C09123=1121.889,263.715,-72.224,-178.349,10.071,149.559
C09124=1121.884,263.963,-72.253,-178.345,10.075,149.559
C09125=1121.880,264.212,-72.283,-178.342,10.077,149.559
C09126=1121.876,264.460,-72.312,-178.338,10.080,149.558
C09127=1121.872,264.708,-72.342,-178.335,10.083,149.558
C09128=1121.868,264.956,-72.371,-178.333,10.085,149.558
C09129=1121.863,265.205,-72.400,-178.330,10.088,149.558
C09130=1121.858,265.453,-72.429,-178.327,10.090,149.558
C09131=1121.854,265.701,-72.458,-178.325,10.093,149.558
C09132=1121.850,265.949,-72.488,-178.323,10.095,149.558
C09133=1121.846,266.198,-72.517,-178.320,10.098,149.558
C09134=1121.842,266.411,-72.542,-178.317,10.100,149.558
C09135=1121.839,266.625,-72.568,-178.315,10.102,149.558
C09136=1121.835,266.838,-72.593,-178.313,10.104,149.557
C09137=1121.832,267.051,-72.619,-178.310,10.106,149.557
C09138=1121.828,267.263,-72.643,-178.308,10.108,149.557
C09139=1121.824,267.477,-72.669,-178.306,10.110,149.557
C09140=1121.821,267.690,-72.694,-178.304,10.112,149.557
C09141=1121.817,267.904,-72.719,-178.302,10.114,149.557
C09142=1121.813,268.152,-72.748,-178.299,10.117,149.557
C09143=1121.809,268.400,-72.778,-178.296,10.119,149.557
C09144=1121.804,268.649,-72.808,-178.293,10.121,149.557
C09145=1121.800,268.897,-72.837,-178.290,10.124,149.557
C09146=1121.795,269.145,-72.867,-178.287,10.127,149.556
C09147=1121.791,269.393,-72.897,-178.285,10.130,149.556
C09148=1121.787,269.641,-72.926,-178.282,10.132,149.556
C09149=1121.783,269.890,-72.956,-178.279,10.134,149.556
C09150=1121.779,270.138,-72.985,-178.276,10.137,149.556
C09151=1121.775,270.386,-73.015,-178.273,10.140,149.556
C09152=1121.771,270.634,-73.044,-178.271,10.142,149.556
C09153=1121.766,270.883,-73.074,-178.268,10.145,149.556
C09154=1121.762,271.131,-73.105,-178.265,10.147,149.556
C09155=1121.758,271.379,-73.134,-178.262,10.150,149.555
C09156=1121.753,271.627,-73.163,-178.259,10.153,149.555
C09157=1121.749,271.875,-73.193,-178.257,10.155,149.555
C09158=1121.745,272.124,-73.222,-178.254,10.158,149.555
C09159=1121.741,272.371,-73.252,-178.251,10.160,149.555
C09160=1121.737,272.620,-73.282,-178.248,10.163,149.555
C09161=1121.732,272.868,-73.312,-178.245,10.166,149.555
C09162=1121.728,273.116,-73.342,-178.242,10.169,149.555
C09163=1121.724,273.364,-73.372,-178.239,10.171,149.555
C09164=1121.720,273.612,-73.401,-178.236,10.174,149.554
C09165=1121.715,273.860,-73.432,-178.233,10.177,149.554
C09166=1121.711,274.109,-73.461,-178.230,10.179,149.554
C09167=1121.707,274.357,-73.491,-178.227,10.182,149.554
C09168=1121.703,274.604,-73.521,-178.224,10.185,149.554
C09169=1121.699,274.853,-73.551,-178.221,10.188,149.554
C09170=1121.694,275.102,-73.581,-178.218,10.190,149.554
C09171=1121.691,275.350,-73.611,-178.215,10.193,149.553
C09172=1121.686,275.598,-73.640,-178.212,10.196,149.553
C09173=1121.682,275.846,-73.671,-178.209,10.198,149.553
C09174=1121.678,276.094,-73.701,-178.206,10.201,149.553
C09175=1121.674,276.342,-73.731,-178.203,10.204,149.553
C09176=1121.669,276.590,-73.761,-178.200,10.206,149.553
C09177=1121.665,276.838,-73.791,-178.197,10.209,149.553
C09178=1121.661,277.087,-73.821,-178.194,10.211,149.552
C09179=1121.657,277.335,-73.852,-178.191,10.214,149.552
C09180=1121.653,277.583,-73.881,-178.188,10.217,149.552
C09181=1121.649,277.831,-73.911,-178.184,10.219,149.552
C09182=1121.644,278.079,-73.941,-178.182,10.222,149.552
C09183=1121.640,278.327,-73.971,-178.178,10.225,149.552
C09184=1121.637,278.575,-74.002,-178.175,10.228,149.551
C09185=1121.632,278.824,-74.032,-178.171,10.231,149.551
C09186=1121.628,279.072,-74.062,-178.168,10.233,149.551
C09187=1121.623,279.320,-74.093,-178.165,10.236,149.551
C09188=1121.619,279.568,-74.122,-178.162,10.238,149.551
C09189=1121.615,279.817,-74.154,-178.158,10.242,149.551
C09190=1121.612,280.029,-74.179,-178.156,10.244,149.550
C09191=1121.608,280.243,-74.205,-178.153,10.246,149.550
C09192=1121.604,280.456,-74.231,-178.151,10.248,149.550
C09193=1121.601,280.669,-74.257,-178.147,10.251,149.550
C09194=1121.597,280.882,-74.283,-178.144,10.254,149.550
C09195=1121.594,281.095,-74.309,-178.142,10.255,149.549
C09196=1121.590,281.308,-74.336,-178.139,10.258,149.549
C09197=1121.583,281.692,-74.383,-178.134,10.262,149.549
C09198=1121.579,281.940,-74.413,-178.131,10.264,149.549
C09199=1121.575,282.189,-74.444,-178.128,10.267,149.549
C09200=1121.571,282.437,-74.475,-178.124,10.270,149.548
C09201=1121.567,282.685,-74.504,-178.121,10.272,149.548
C09202=1121.562,282.933,-74.535,-178.119,10.275,149.548
C09203=1121.559,283.181,-74.565,-178.115,10.277,149.548
C09204=1121.554,283.429,-74.596,-178.113,10.279,149.548
C09205=1121.550,283.677,-74.626,-178.110,10.282,149.548
C09206=1121.546,283.925,-74.657,-178.107,10.285,149.547
C09207=1121.542,284.173,-74.688,-178.103,10.287,149.547
C09208=1121.538,284.421,-74.718,-178.100,10.290,149.547
C09209=1121.533,284.669,-74.749,-178.097,10.293,149.547
C09210=1121.529,284.918,-74.780,-178.094,10.295,149.547
C09211=1121.525,285.165,-74.810,-178.091,10.298,149.547
C09212=1121.521,285.413,-74.841,-178.088,10.300,149.546
C09213=1121.517,285.662,-74.872,-178.085,10.303,149.546
C09214=1121.513,285.910,-74.902,-178.082,10.305,149.546
C09215=1121.508,286.158,-74.933,-178.079,10.307,149.546
C09216=1121.504,286.406,-74.964,-178.076,10.310,149.546
C09217=1121.500,286.654,-74.995,-178.073,10.313,149.546
C09218=1121.496,286.902,-75.025,-178.070,10.315,149.545
C09219=1121.492,287.150,-75.056,-178.067,10.318,149.545
C09220=1121.488,287.398,-75.087,-178.064,10.320,149.545
C09221=1121.483,287.646,-75.117,-178.060,10.323,149.545
C09222=1121.479,287.894,-75.149,-178.057,10.326,149.545
C09223=1121.475,288.142,-75.180,-178.055,10.327,149.544
C09224=1121.471,288.390,-75.210,-178.052,10.330,149.544
C09225=1121.467,288.638,-75.241,-178.049,10.333,149.544
C09226=1121.462,288.886,-75.272,-178.045,10.335,149.544
C09227=1121.458,289.135,-75.303,-178.043,10.338,149.544
C09228=1121.455,289.382,-75.334,-178.039,10.340,149.544
C09229=1121.451,289.631,-75.365,-178.036,10.343,149.543
C09230=1121.446,289.879,-75.396,-178.033,10.346,149.543
C09231=1121.441,290.127,-75.427,-178.030,10.348,149.543
C09232=1121.438,290.375,-75.459,-178.027,10.351,149.543
C09233=1121.433,290.623,-75.489,-178.024,10.353,149.543
C09234=1121.430,290.871,-75.520,-178.021,10.356,149.543
C09235=1121.426,291.118,-75.551,-178.018,10.358,149.542
C09236=1121.422,291.367,-75.582,-178.015,10.361,149.542
C09237=1121.417,291.615,-75.613,-178.012,10.363,149.542
C09238=1121.413,291.863,-75.645,-178.009,10.366,149.542
C09239=1121.409,292.111,-75.676,-178.006,10.368,149.542
C09240=1121.405,292.360,-75.707,-178.003,10.371,149.542
C09241=1121.401,292.607,-75.738,-177.999,10.374,149.541
C09242=1121.397,292.855,-75.769,-177.996,10.376,149.541
C09243=1121.393,293.103,-75.800,-177.994,10.378,149.541
C09244=1121.389,293.351,-75.832,-177.991,10.381,149.541
C09245=1121.384,293.599,-75.863,-177.987,10.383,149.541
C09246=1121.378,293.982,-75.912,-177.983,10.387,149.540
C09247=1121.371,294.365,-75.959,-177.978,10.391,149.540
C09248=1121.365,294.749,-76.008,-177.974,10.395,149.540
C09249=1121.359,295.132,-76.056,-177.969,10.399,149.539
C09250=1121.354,295.379,-76.088,-177.966,10.401,149.539
C09251=1121.351,295.627,-76.119,-177.962,10.404,149.539
C09252=1121.346,295.875,-76.150,-177.959,10.407,149.539
C09253=1121.342,296.123,-76.182,-177.956,10.409,149.539
C09254=1121.338,296.372,-76.213,-177.953,10.412,149.539
C09255=1121.334,296.619,-76.245,-177.950,10.414,149.538
C09256=1121.330,296.868,-76.277,-177.947,10.417,149.538
C09257=1121.326,297.115,-76.307,-177.943,10.419,149.538
C09258=1121.322,297.364,-76.339,-177.941,10.422,149.538
C09259=1121.318,297.611,-76.371,-177.938,10.424,149.538
C09260=1121.313,297.860,-76.402,-177.935,10.427,149.538
C09261=1121.309,298.108,-76.434,-177.932,10.429,149.537
C09262=1121.305,298.355,-76.466,-177.929,10.432,149.537
C09263=1121.301,298.604,-76.497,-177.925,10.434,149.537
C09264=1121.297,298.851,-76.528,-177.922,10.437,149.537
C09265=1121.293,299.099,-76.560,-177.919,10.439,149.537
C09266=1121.289,299.347,-76.592,-177.916,10.442,149.537
C09267=1121.285,299.595,-76.623,-177.913,10.445,149.536
C09268=1121.280,299.844,-76.655,-177.910,10.447,149.536
C09269=1121.277,300.092,-76.687,-177.906,10.450,149.536
C09270=1121.272,300.339,-76.719,-177.904,10.452,149.536
C09271=1121.269,300.587,-76.750,-177.901,10.454,149.536
C09272=1121.265,300.835,-76.782,-177.898,10.457,149.535
C09273=1121.260,301.083,-76.814,-177.895,10.459,149.535
C09274=1121.256,301.331,-76.846,-177.892,10.462,149.535
C09275=1121.252,301.579,-76.877,-177.888,10.465,149.535
C09276=1121.248,301.827,-76.909,-177.885,10.467,149.535
C09277=1121.243,302.075,-76.941,-177.882,10.470,149.534
C09278=1121.240,302.323,-76.973,-177.879,10.473,149.534
C09279=1121.235,302.570,-77.004,-177.876,10.475,149.534
C09280=1121.232,302.818,-77.036,-177.873,10.478,149.534
C09281=1121.227,303.067,-77.069,-177.870,10.480,149.534
C09282=1121.223,303.314,-77.100,-177.867,10.482,149.534
C09283=1121.219,303.562,-77.132,-177.864,10.485,149.533
C09284=1121.215,303.811,-77.165,-177.861,10.487,149.533
C09285=1121.210,304.058,-77.196,-177.858,10.490,149.533
C09286=1121.207,304.306,-77.228,-177.855,10.493,149.533
C09287=1121.202,304.554,-77.260,-177.851,10.495,149.533
C09288=1121.199,304.802,-77.293,-177.848,10.498,149.533
C09289=1121.195,305.049,-77.324,-177.845,10.500,149.532
C09290=1121.190,305.297,-77.357,-177.842,10.503,149.532
C09291=1121.186,305.545,-77.389,-177.839,10.506,149.532
C09292=1121.182,305.794,-77.421,-177.836,10.508,149.532
C09293=1121.178,306.041,-77.453,-177.833,10.510,149.532
C09294=1121.174,306.289,-77.484,-177.830,10.512,149.531
C09295=1121.170,306.537,-77.518,-177.827,10.515,149.531
C09296=1121.166,306.785,-77.549,-177.824,10.518,149.531
C09297=1121.162,307.033,-77.582,-177.821,10.520,149.531
C09298=1121.158,307.246,-77.609,-177.818,10.522,149.531
C09299=1121.155,307.459,-77.637,-177.815,10.525,149.531
C09300=1121.151,307.671,-77.664,-177.813,10.527,149.531
C09301=1121.148,307.884,-77.693,-177.809,10.529,149.530
C09302=1121.144,308.097,-77.720,-177.807,10.531,149.530
C09303=1121.141,308.310,-77.747,-177.805,10.533,149.530
C09304=1121.137,308.522,-77.775,-177.802,10.536,149.530
C09305=1121.133,308.736,-77.803,-177.799,10.538,149.530
C09306=1121.130,308.983,-77.835,-177.796,10.540,149.530
C09307=1121.125,309.232,-77.868,-177.793,10.543,149.529
C09308=1121.121,309.479,-77.899,-177.790,10.545,149.529
C09309=1121.117,309.727,-77.933,-177.787,10.548,149.529
C09310=1121.113,309.975,-77.964,-177.783,10.550,149.529
C09311=1121.109,310.223,-77.998,-177.780,10.553,149.529
C09312=1121.105,310.471,-78.029,-177.778,10.555,149.528
C09313=1121.101,310.719,-78.062,-177.775,10.558,149.528
C09314=1121.098,310.966,-78.094,-177.771,10.560,149.528
C09315=1121.093,311.214,-78.126,-177.768,10.563,149.528
C09316=1121.088,311.462,-78.160,-177.765,10.565,149.528
C09317=1121.085,311.710,-78.191,-177.762,10.568,149.528
C09318=1121.081,311.958,-78.225,-177.759,10.571,149.527
C09319=1121.077,312.206,-78.256,-177.756,10.573,149.527
C09320=1121.073,312.453,-78.290,-177.753,10.576,149.527
C09321=1121.068,312.702,-78.322,-177.749,10.578,149.527
C09322=1121.065,312.949,-78.355,-177.746,10.581,149.527
C09323=1121.061,313.197,-78.388,-177.743,10.583,149.527
C09324=1121.057,313.445,-78.420,-177.740,10.586,149.526
C09325=1121.053,313.693,-78.453,-177.738,10.588,149.526
C09326=1121.048,313.941,-78.485,-177.734,10.590,149.526
C09327=1121.044,314.188,-78.517,-177.731,10.593,149.526
C09328=1121.040,314.435,-78.551,-177.728,10.595,149.526
C09329=1121.036,314.684,-78.583,-177.725,10.598,149.525
C09330=1121.032,314.931,-78.616,-177.722,10.601,149.525
C09331=1121.028,315.179,-78.649,-177.718,10.603,149.525
C09332=1121.024,315.427,-78.681,-177.715,10.606,149.525
C09333=1121.020,315.675,-78.714,-177.712,10.608,149.525
C09334=1121.016,315.922,-78.747,-177.709,10.611,149.524
C09335=1121.012,316.171,-78.779,-177.706,10.614,149.524
C09336=1121.008,316.418,-78.812,-177.703,10.616,149.524
C09337=1121.004,316.666,-78.846,-177.700,10.618,149.524
C09338=1121.000,316.914,-78.878,-177.697,10.620,149.524
C09339=1120.996,317.161,-78.911,-177.694,10.623,149.524
C09340=1120.992,317.410,-78.944,-177.691,10.626,149.523
C09341=1120.988,317.657,-78.977,-177.687,10.628,149.523
C09342=1120.984,317.905,-79.009,-177.684,10.631,149.523
C09343=1120.980,318.153,-79.043,-177.681,10.633,149.523
C09344=1120.976,318.401,-79.076,-177.678,10.636,149.523
C09345=1120.972,318.649,-79.109,-177.674,10.638,149.522
C09346=1120.968,318.896,-79.142,-177.671,10.641,149.522
C09347=1120.964,319.144,-79.176,-177.668,10.643,149.522
C09348=1120.960,319.392,-79.207,-177.665,10.646,149.522
C09349=1120.956,319.640,-79.241,-177.662,10.649,149.522
C09350=1120.952,319.888,-79.274,-177.659,10.650,149.521
C09351=1120.948,320.135,-79.307,-177.656,10.653,149.521
C09352=1120.944,320.383,-79.340,-177.653,10.656,149.521
C09353=1120.940,320.631,-79.373,-177.650,10.658,149.521
C09354=1120.937,320.843,-79.402,-177.647,10.661,149.521
C09355=1120.933,321.056,-79.430,-177.644,10.663,149.521
C09356=1120.929,321.268,-79.459,-177.642,10.664,149.520
C09357=1120.926,321.481,-79.487,-177.639,10.667,149.520
C09358=1120.923,321.694,-79.516,-177.636,10.669,149.520
C09359=1120.920,321.907,-79.544,-177.634,10.671,149.520
C09360=1120.916,322.120,-79.573,-177.631,10.674,149.520
C09361=1120.912,322.332,-79.601,-177.628,10.675,149.520
C09362=1120.909,322.581,-79.635,-177.625,10.678,149.520
C09363=1120.905,322.828,-79.668,-177.622,10.680,149.519
C09364=1120.901,323.075,-79.702,-177.619,10.683,149.519
C09365=1120.897,323.323,-79.735,-177.616,10.686,149.519
C09366=1120.892,323.571,-79.768,-177.612,10.688,149.519
C09367=1120.888,323.819,-79.801,-177.609,10.691,149.519
C09368=1120.885,324.067,-79.835,-177.606,10.693,149.518
C09369=1120.881,324.314,-79.868,-177.603,10.696,149.518
C09370=1120.877,324.562,-79.902,-177.599,10.698,149.518
C09371=1120.873,324.810,-79.935,-177.597,10.701,149.518
C09372=1120.868,325.057,-79.968,-177.594,10.703,149.518
C09373=1120.865,325.304,-80.002,-177.591,10.705,149.517
C09374=1120.861,325.553,-80.035,-177.588,10.708,149.517
C09375=1120.857,325.801,-80.069,-177.584,10.710,149.517
C09376=1120.853,326.048,-80.102,-177.581,10.713,149.517
C09377=1120.849,326.295,-80.136,-177.578,10.716,149.517
C09378=1120.845,326.543,-80.169,-177.575,10.718,149.517
C09379=1120.841,326.792,-80.202,-177.571,10.721,149.516
C09380=1120.837,327.039,-80.237,-177.568,10.723,149.516
C09381=1120.833,327.287,-80.270,-177.565,10.726,149.516
C09382=1120.829,327.534,-80.304,-177.562,10.728,149.516
C09383=1120.825,327.782,-80.337,-177.559,10.731,149.515
C09384=1120.821,328.030,-80.370,-177.556,10.733,149.515
C09385=1120.817,328.277,-80.404,-177.553,10.735,149.515
C09386=1120.812,328.525,-80.438,-177.550,10.738,149.515
C09387=1120.809,328.773,-80.472,-177.547,10.740,149.515
C09388=1120.805,329.021,-80.505,-177.543,10.743,149.515
C09389=1120.801,329.268,-80.539,-177.540,10.745,149.514
C09390=1120.797,329.516,-80.572,-177.537,10.748,149.514
C09391=1120.793,329.764,-80.607,-177.534,10.750,149.514
C09392=1120.789,330.011,-80.640,-177.530,10.753,149.514
C09393=1120.785,330.259,-80.674,-177.527,10.755,149.514
C09394=1120.782,330.507,-80.708,-177.524,10.758,149.514
C09395=1120.777,330.754,-80.742,-177.521,10.761,149.513
C09396=1120.773,331.001,-80.776,-177.518,10.763,149.513
C09397=1120.770,331.250,-80.810,-177.515,10.766,149.513
C09398=1120.766,331.497,-80.844,-177.511,10.768,149.513
C09399=1120.761,331.745,-80.877,-177.508,10.771,149.512
C09400=1120.758,331.993,-80.912,-177.505,10.772,149.512
C09401=1120.754,332.240,-80.945,-177.502,10.775,149.512
C09402=1120.749,332.488,-80.979,-177.499,10.778,149.512
C09403=1120.746,332.736,-81.013,-177.496,10.780,149.512
C09404=1120.742,332.983,-81.047,-177.493,10.783,149.512
C09405=1120.737,333.230,-81.082,-177.490,10.785,149.511
C09406=1120.734,333.479,-81.115,-177.486,10.788,149.511
C09407=1120.730,333.726,-81.149,-177.483,10.790,149.511
C09408=1120.725,333.973,-81.184,-177.480,10.793,149.511
C09409=1120.722,334.221,-81.218,-177.477,10.795,149.511
C09410=1120.719,334.434,-81.247,-177.474,10.797,149.510
C09411=1120.715,334.646,-81.276,-177.471,10.800,149.510
C09412=1120.712,334.859,-81.305,-177.468,10.802,149.510
C09413=1120.709,335.071,-81.335,-177.466,10.804,149.510
C09414=1120.705,335.284,-81.364,-177.463,10.806,149.510
C09415=1120.702,335.497,-81.393,-177.460,10.808,149.510
C09416=1120.698,335.709,-81.422,-177.458,10.810,149.509
C09417=1120.695,335.922,-81.452,-177.455,10.812,149.509
C09418=1120.691,336.169,-81.486,-177.452,10.815,149.509
C09419=1120.687,336.417,-81.520,-177.448,10.817,149.509
C09420=1120.683,336.664,-81.555,-177.445,10.820,149.509
C09421=1120.679,336.911,-81.589,-177.442,10.823,149.509
C09422=1120.675,337.160,-81.624,-177.439,10.824,149.508
C09423=1120.671,337.407,-81.658,-177.436,10.827,149.508
C09424=1120.667,337.655,-81.692,-177.433,10.830,149.508
C09425=1120.663,337.902,-81.726,-177.430,10.832,149.508
C09426=1120.660,338.150,-81.761,-177.426,10.834,149.507
C09427=1120.656,338.397,-81.795,-177.423,10.837,149.507
C09428=1120.652,338.645,-81.830,-177.420,10.839,149.507
C09429=1120.647,338.893,-81.864,-177.417,10.842,149.507
C09430=1120.644,339.140,-81.898,-177.414,10.845,149.507
C09431=1120.639,339.388,-81.933,-177.410,10.847,149.506
C09432=1120.636,339.636,-81.967,-177.407,10.849,149.506
C09433=1120.632,339.883,-82.002,-177.404,10.852,149.506
C09434=1120.628,340.131,-82.036,-177.401,10.855,149.506
C09435=1120.624,340.378,-82.070,-177.397,10.857,149.506
C09436=1120.620,340.626,-82.105,-177.394,10.860,149.506
C09437=1120.616,340.873,-82.140,-177.391,10.861,149.505
C09438=1120.612,341.121,-82.175,-177.388,10.864,149.505
C09439=1120.608,341.368,-82.209,-177.385,10.867,149.505
C09440=1120.604,341.616,-82.243,-177.382,10.869,149.505
C09441=1120.600,341.864,-82.278,-177.378,10.871,149.504
C09442=1120.596,342.111,-82.313,-177.375,10.874,149.504
C09443=1120.592,342.358,-82.347,-177.372,10.877,149.504
C09444=1120.588,342.606,-82.382,-177.369,10.879,149.504
C09445=1120.584,342.854,-82.416,-177.366,10.882,149.504
C09446=1120.580,343.101,-82.452,-177.362,10.884,149.504
C09447=1120.577,343.349,-82.486,-177.359,10.887,149.503
C09448=1120.572,343.597,-82.521,-177.356,10.889,149.503
C09449=1120.569,343.844,-82.556,-177.353,10.892,149.503
C09450=1120.564,344.092,-82.591,-177.349,10.894,149.503
C09451=1120.561,344.339,-82.625,-177.346,10.897,149.503
C09452=1120.557,344.587,-82.661,-177.343,10.898,149.502
C09453=1120.553,344.834,-82.695,-177.340,10.901,149.502
C09454=1120.549,345.082,-82.730,-177.337,10.904,149.502
C09455=1120.545,345.329,-82.764,-177.334,10.906,149.502
C09456=1120.541,345.577,-82.799,-177.331,10.909,149.502
C09457=1120.538,345.824,-82.835,-177.327,10.911,149.501
C09458=1120.533,346.072,-82.869,-177.324,10.913,149.501
C09459=1120.529,346.319,-82.905,-177.321,10.916,149.501
C09460=1120.526,346.567,-82.939,-177.318,10.919,149.501
C09461=1120.522,346.814,-82.974,-177.314,10.921,149.501
C09462=1120.518,347.062,-83.009,-177.311,10.924,149.500
C09463=1120.514,347.309,-83.044,-177.308,10.926,149.500
C09464=1120.510,347.557,-83.079,-177.305,10.929,149.500
C09465=1120.506,347.805,-83.115,-177.301,10.931,149.500
C09466=1120.503,348.017,-83.144,-177.299,10.933,149.500
C09467=1120.499,348.229,-83.174,-177.296,10.935,149.499
C09468=1120.496,348.441,-83.205,-177.293,10.937,149.499
C09469=1120.493,348.654,-83.235,-177.291,10.939,149.499
C09470=1120.489,348.867,-83.265,-177.288,10.941,149.499
C09471=1120.486,349.079,-83.294,-177.285,10.944,149.499
C09472=1120.482,349.291,-83.325,-177.282,10.945,149.498
C09473=1120.480,349.504,-83.355,-177.279,10.948,149.498
C09474=1120.476,349.750,-83.391,-177.276,10.950,149.498
C09475=1120.472,349.999,-83.425,-177.272,10.953,149.498
C09476=1120.468,350.246,-83.461,-177.269,10.955,149.498
C09477=1120.464,350.494,-83.496,-177.266,10.958,149.497
C09478=1120.460,350.741,-83.531,-177.262,10.961,149.497
C09479=1120.456,350.989,-83.566,-177.259,10.963,149.497
C09480=1120.452,351.236,-83.602,-177.255,10.966,149.497
C09481=1120.449,351.484,-83.638,-177.252,10.968,149.496
C09482=1120.445,351.730,-83.673,-177.248,10.970,149.496
C09483=1120.441,351.978,-83.708,-177.244,10.974,149.496
C09484=1120.437,352.226,-83.743,-177.241,10.976,149.496
C09485=1120.433,352.473,-83.779,-177.238,10.979,149.495
C09486=1120.429,352.720,-83.814,-177.234,10.981,149.495
C09487=1120.425,352.968,-83.849,-177.231,10.983,149.495
C09488=1120.422,353.215,-83.885,-177.228,10.986,149.495
C09489=1120.418,353.463,-83.921,-177.223,10.989,149.494
C09490=1120.414,353.711,-83.957,-177.220,10.991,149.494
C09491=1120.409,353.957,-83.992,-177.217,10.994,149.494
C09492=1120.406,354.205,-84.027,-177.213,10.996,149.494
C09493=1120.402,354.453,-84.062,-177.210,10.999,149.493
C09494=1120.398,354.700,-84.098,-177.206,11.001,149.493
C09495=1120.394,354.948,-84.133,-177.203,11.003,149.493
C09496=1120.391,355.195,-84.169,-177.200,11.006,149.493
C09497=1120.387,355.442,-84.205,-177.197,11.008,149.492
C09498=1120.383,355.689,-84.240,-177.193,11.011,149.492
C09499=1120.379,355.937,-84.276,-177.189,11.014,149.492
C09500=1120.375,356.184,-84.312,-177.186,11.016,149.492
C09501=1120.371,356.432,-84.348,-177.182,11.019,149.491
C09502=1120.368,356.679,-84.383,-177.179,11.021,149.491
C09503=1120.364,356.927,-84.419,-177.176,11.023,149.491
C09504=1120.360,357.175,-84.455,-177.172,11.026,149.491
C09505=1120.356,357.422,-84.490,-177.169,11.028,149.490
C09506=1120.353,357.669,-84.527,-177.165,11.031,149.490
C09507=1120.348,357.916,-84.562,-177.162,11.033,149.490
C09508=1120.345,358.163,-84.597,-177.158,11.035,149.489
C09509=1120.340,358.411,-84.633,-177.155,11.038,149.489
C09510=1120.337,358.659,-84.669,-177.152,11.040,149.489
C09511=1120.333,358.906,-84.705,-177.148,11.043,149.489
C09512=1120.330,359.153,-84.741,-177.145,11.045,149.489
C09513=1120.325,359.401,-84.777,-177.141,11.047,149.488
C09514=1120.322,359.648,-84.813,-177.138,11.050,149.488
C09515=1120.318,359.895,-84.849,-177.135,11.052,149.488
C09516=1120.314,360.143,-84.885,-177.131,11.055,149.488
C09517=1120.310,360.391,-84.920,-177.128,11.057,149.487
C09518=1120.307,360.638,-84.957,-177.124,11.059,149.487
C09519=1120.302,360.885,-84.993,-177.121,11.062,149.487
C09520=1120.299,361.132,-85.029,-177.118,11.064,149.486
C09521=1120.295,361.380,-85.065,-177.115,11.067,149.486
C09522=1120.292,361.592,-85.096,-177.111,11.069,149.486
C09523=1120.289,361.804,-85.127,-177.109,11.071,149.486
C09524=1120.285,362.016,-85.158,-177.105,11.073,149.486
C09525=1120.282,362.229,-85.189,-177.103,11.075,149.485
C09526=1120.279,362.441,-85.219,-177.100,11.077,149.485
C09527=1120.276,362.653,-85.251,-177.097,11.079,149.485
C09528=1120.272,362.865,-85.282,-177.094,11.081,149.485
C09529=1120.269,363.078,-85.313,-177.091,11.083,149.484
C09530=1120.266,363.325,-85.348,-177.087,11.086,149.484
C09531=1120.262,363.572,-85.385,-177.084,11.088,149.484
C09532=1120.258,363.819,-85.421,-177.081,11.091,149.484
C09533=1120.254,364.067,-85.458,-177.077,11.093,149.484
C09534=1120.250,364.314,-85.494,-177.074,11.094,149.483
C09535=1120.246,364.562,-85.530,-177.071,11.097,149.483
C09536=1120.243,364.809,-85.566,-177.068,11.099,149.483
C09537=1120.239,365.056,-85.603,-177.064,11.102,149.482
C09538=1120.235,365.303,-85.639,-177.061,11.104,149.482
C09539=1120.231,365.551,-85.676,-177.057,11.106,149.482
C09540=1120.227,365.798,-85.711,-177.054,11.109,149.482
C09541=1120.224,366.046,-85.748,-177.051,11.111,149.481
C09542=1120.220,366.293,-85.785,-177.048,11.114,149.481
C09543=1120.216,366.540,-85.821,-177.044,11.116,149.481
C09544=1120.213,366.788,-85.857,-177.041,11.119,149.481
C09545=1120.208,367.035,-85.894,-177.038,11.121,149.481
C09546=1120.204,367.282,-85.931,-177.034,11.123,149.480
C09547=1120.201,367.529,-85.967,-177.031,11.126,149.480
C09548=1120.197,367.777,-86.003,-177.028,11.128,149.480
C09549=1120.193,368.024,-86.039,-177.025,11.130,149.480
C09550=1120.190,368.271,-86.077,-177.021,11.133,149.479
C09551=1120.186,368.519,-86.113,-177.018,11.135,149.479
C09552=1120.182,368.766,-86.150,-177.015,11.138,149.479
C09553=1120.178,369.013,-86.186,-177.011,11.140,149.479
C09554=1120.175,369.260,-86.222,-177.008,11.142,149.478
C09555=1120.170,369.507,-86.259,-177.005,11.145,149.478
C09556=1120.167,369.755,-86.296,-177.001,11.147,149.478
C09557=1120.164,370.002,-86.332,-176.998,11.149,149.478
C09558=1120.160,370.249,-86.369,-176.995,11.151,149.477
C09559=1120.155,370.497,-86.406,-176.992,11.154,149.477
C09560=1120.151,370.744,-86.443,-176.989,11.156,149.477
C09561=1120.149,370.991,-86.480,-176.985,11.159,149.477
C09562=1120.144,371.239,-86.517,-176.982,11.161,149.477
C09563=1120.140,371.486,-86.553,-176.979,11.164,149.476
C09564=1120.137,371.733,-86.590,-176.975,11.166,149.476
C09565=1120.133,371.980,-86.627,-176.972,11.169,149.476
C09566=1120.129,372.228,-86.664,-176.969,11.170,149.476
C09567=1120.125,372.475,-86.701,-176.966,11.173,149.476
C09568=1120.122,372.722,-86.737,-176.963,11.175,149.475
C09569=1120.118,372.969,-86.774,-176.960,11.178,149.475
C09570=1120.114,373.217,-86.811,-176.956,11.180,149.475
C09571=1120.110,373.464,-86.848,-176.953,11.183,149.475
C09572=1120.107,373.711,-86.884,-176.950,11.186,149.475
C09573=1120.103,373.957,-86.922,-176.947,11.187,149.474
C09574=1120.100,374.205,-86.959,-176.944,11.190,149.474
C09575=1120.096,374.453,-86.996,-176.941,11.192,149.474
C09576=1120.091,374.700,-87.033,-176.937,11.195,149.474
C09577=1120.087,374.947,-87.069,-176.934,11.197,149.474
C09578=1120.085,375.159,-87.101,-176.932,11.199,149.473
C09579=1120.082,375.371,-87.133,-176.929,11.202,149.473
C09580=1120.078,375.583,-87.164,-176.926,11.203,149.473
C09581=1120.075,375.795,-87.197,-176.924,11.205,149.473
C09582=1120.072,376.007,-87.229,-176.921,11.207,149.473
C09583=1120.069,376.220,-87.260,-176.918,11.210,149.473
C09584=1120.066,376.431,-87.292,-176.915,11.212,149.473
C09585=1120.062,376.644,-87.324,-176.913,11.214,149.473
C09586=1120.058,376.891,-87.361,-176.910,11.216,149.472
C09587=1120.055,377.139,-87.398,-176.907,11.219,149.472
C09588=1120.052,377.385,-87.435,-176.903,11.221,149.472
C09589=1120.047,377.632,-87.472,-176.900,11.224,149.472
C09590=1120.044,377.880,-87.510,-176.897,11.226,149.472
C09591=1120.040,378.127,-87.547,-176.894,11.229,149.471
C09592=1120.036,378.374,-87.584,-176.891,11.231,149.471
C09593=1120.033,378.621,-87.622,-176.888,11.233,149.471
C09594=1120.029,378.868,-87.659,-176.885,11.236,149.471
C09595=1120.025,379.115,-87.696,-176.882,11.239,149.471
C09596=1120.022,379.363,-87.734,-176.879,11.241,149.471
C09597=1120.017,379.610,-87.770,-176.875,11.244,149.471
C09598=1120.014,379.857,-87.808,-176.873,11.246,149.471
C09599=1120.010,380.104,-87.845,-176.870,11.248,149.470
C09600=1120.006,380.351,-87.883,-176.867,11.251,149.470
C09601=1120.003,380.599,-87.920,-176.864,11.253,149.470
C09602=1119.999,380.845,-87.958,-176.860,11.256,149.470
C09603=1119.996,381.093,-87.995,-176.857,11.259,149.470
C09604=1119.992,381.340,-88.032,-176.854,11.261,149.470
C09605=1119.987,381.587,-88.071,-176.852,11.263,149.470
C09606=1119.984,381.835,-88.108,-176.849,11.266,149.470
C09607=1119.980,382.081,-88.145,-176.846,11.269,149.469
C09608=1119.976,382.329,-88.183,-176.842,11.271,149.469
C09609=1119.973,382.576,-88.220,-176.840,11.274,149.469
C09610=1119.969,382.823,-88.258,-176.837,11.277,149.469
C09611=1119.965,383.070,-88.295,-176.833,11.279,149.469
C09612=1119.962,383.317,-88.333,-176.831,11.281,149.469
C09613=1119.958,383.564,-88.370,-176.828,11.284,149.469
C09614=1119.954,383.811,-88.407,-176.826,11.286,149.469
C09615=1119.950,384.059,-88.446,-176.824,11.288,149.469
C09616=1119.947,384.305,-88.483,-176.822,11.290,149.469
C09617=1119.943,384.553,-88.521,-176.820,11.293,149.469
C09618=1119.939,384.800,-88.558,-176.818,11.295,149.469
C09619=1119.936,385.047,-88.596,-176.816,11.297,149.469
C09620=1119.932,385.294,-88.634,-176.813,11.299,149.469
C09621=1119.928,385.541,-88.672,-176.812,11.302,149.469
C09622=1119.924,385.788,-88.709,-176.809,11.304,149.469
C09623=1119.921,386.036,-88.747,-176.807,11.306,149.469
C09624=1119.917,386.282,-88.785,-176.806,11.308,149.470
C09625=1119.914,386.529,-88.823,-176.803,11.310,149.470
C09626=1119.910,386.776,-88.861,-176.801,11.313,149.470
C09627=1119.906,387.024,-88.899,-176.800,11.315,149.470
C09628=1119.902,387.271,-88.936,-176.798,11.317,149.470
C09629=1119.899,387.518,-88.974,-176.796,11.320,149.470
C09630=1119.895,387.765,-89.011,-176.794,11.322,149.470
C09631=1119.891,388.012,-89.050,-176.791,11.325,149.470
C09632=1119.888,388.260,-89.088,-176.790,11.328,149.471
C09633=1119.884,388.506,-89.125,-176.788,11.330,149.471
C09634=1119.881,388.718,-89.158,-176.786,11.332,149.471
C09635=1119.878,388.930,-89.190,-176.785,11.334,149.471
C09636=1119.875,389.142,-89.223,-176.783,11.336,149.471
C09637=1119.872,389.354,-89.255,-176.781,11.339,149.471
C09638=1119.868,389.566,-89.287,-176.780,11.341,149.471
C09639=1119.865,389.778,-89.321,-176.778,11.343,149.472
C09640=1119.862,389.990,-89.353,-176.776,11.345,149.472
C09641=1119.859,390.202,-89.385,-176.775,11.348,149.472
C09642=1119.856,390.449,-89.423,-176.773,11.350,149.472
C09643=1119.852,390.696,-89.461,-176.771,11.353,149.472
C09644=1119.848,390.943,-89.499,-176.769,11.355,149.473
C09645=1119.845,391.191,-89.537,-176.768,11.358,149.473
C09646=1119.841,391.437,-89.575,-176.766,11.361,149.473
C09647=1119.837,391.685,-89.613,-176.764,11.364,149.473
C09648=1119.833,391.931,-89.651,-176.762,11.366,149.474
C09649=1119.830,392.179,-89.689,-176.760,11.370,149.474
C09650=1119.826,392.426,-89.727,-176.759,11.372,149.474
C09651=1119.823,392.672,-89.766,-176.757,11.375,149.475
C09652=1119.820,392.919,-89.803,-176.755,11.378,149.475
C09653=1119.815,393.166,-89.842,-176.753,11.381,149.475
C09654=1119.812,393.414,-89.880,-176.752,11.384,149.475
C09655=1119.808,393.661,-89.918,-176.750,11.387,149.476
C09656=1119.804,393.908,-89.956,-176.748,11.390,149.476
C09657=1119.801,394.155,-89.994,-176.747,11.392,149.476
C09658=1119.796,394.402,-90.032,-176.744,11.396,149.477
C09659=1119.794,394.648,-90.070,-176.743,11.399,149.477
C09660=1119.790,394.896,-90.109,-176.742,11.402,149.478
C09661=1119.786,395.143,-90.147,-176.740,11.405,149.478
C09662=1119.783,395.390,-90.185,-176.739,11.408,149.478
C09663=1119.779,395.637,-90.223,-176.737,11.412,149.479
C09664=1119.775,395.883,-90.261,-176.735,11.414,149.479
C09665=1119.771,396.131,-90.300,-176.733,11.418,149.480
C09666=1119.768,396.378,-90.338,-176.732,11.421,149.480
C09667=1119.764,396.625,-90.376,-176.730,11.425,149.481
C09668=1119.761,396.872,-90.415,-176.729,11.428,149.481
C09669=1119.757,397.119,-90.453,-176.727,11.431,149.481
C09670=1119.753,397.366,-90.491,-176.726,11.434,149.482
C09671=1119.749,397.614,-90.529,-176.724,11.438,149.483
C09672=1119.746,397.860,-90.568,-176.723,11.441,149.483
C09673=1119.742,398.107,-90.606,-176.721,11.444,149.483
C09674=1119.738,398.354,-90.644,-176.719,11.448,149.484
C09675=1119.735,398.601,-90.683,-176.718,11.451,149.484
C09676=1119.732,398.849,-90.721,-176.716,11.455,149.485
C09677=1119.727,399.095,-90.759,-176.716,11.458,149.486
C09678=1119.724,399.342,-90.798,-176.714,11.462,149.486
C09679=1119.720,399.590,-90.837,-176.712,11.466,149.487
C09680=1119.717,399.836,-90.875,-176.711,11.469,149.487
C09681=1119.713,400.083,-90.913,-176.709,11.473,149.488
C09682=1119.710,400.331,-90.951,-176.708,11.477,149.489
C09683=1119.706,400.577,-90.991,-176.707,11.480,149.489
C09684=1119.702,400.824,-91.028,-176.706,11.484,149.490
C09685=1119.699,401.071,-91.067,-176.704,11.488,149.490
C09686=1119.695,401.319,-91.106,-176.703,11.492,149.491
C09687=1119.692,401.565,-91.145,-176.702,11.495,149.492
C09688=1119.687,401.812,-91.183,-176.700,11.499,149.492
C09689=1119.684,402.059,-91.221,-176.699,11.503,149.493
C09690=1119.681,402.271,-91.254,-176.698,11.506,149.494
C09691=1119.678,402.483,-91.287,-176.697,11.509,149.494
C09692=1119.675,402.695,-91.321,-176.695,11.513,149.495
C09693=1119.672,402.906,-91.354,-176.695,11.517,149.496
C09694=1119.668,403.118,-91.387,-176.694,11.520,149.496
C09695=1119.665,403.330,-91.421,-176.692,11.524,149.497
C09696=1119.662,403.542,-91.453,-176.692,11.527,149.498
C09697=1119.659,403.753,-91.486,-176.691,11.530,149.498
C09698=1119.656,404.000,-91.525,-176.690,11.535,149.499
C09699=1119.652,404.248,-91.564,-176.688,11.539,149.500
C09700=1119.649,404.495,-91.602,-176.687,11.543,149.500
C09701=1119.645,404.742,-91.642,-176.686,11.547,149.501
C09702=1119.641,404.988,-91.680,-176.685,11.551,149.502
C09703=1119.638,405.235,-91.718,-176.684,11.556,149.503
C09704=1119.634,405.482,-91.758,-176.682,11.560,149.504
C09705=1119.630,405.730,-91.796,-176.681,11.564,149.505
C09706=1119.627,405.976,-91.835,-176.680,11.569,149.506
C09707=1119.623,406.223,-91.874,-176.679,11.573,149.506
C09708=1119.619,406.470,-91.912,-176.678,11.577,149.507
C09709=1119.616,406.717,-91.951,-176.677,11.582,149.508
C09710=1119.613,406.964,-91.990,-176.676,11.586,149.509
C09711=1119.609,407.211,-92.029,-176.675,11.591,149.510
C09712=1119.605,407.458,-92.068,-176.674,11.595,149.511
C09713=1119.602,407.705,-92.107,-176.673,11.600,149.512
C09714=1119.598,407.951,-92.145,-176.672,11.604,149.513
C09715=1119.594,408.199,-92.184,-176.671,11.610,149.514
C09716=1119.591,408.445,-92.223,-176.670,11.614,149.515
C09717=1119.588,408.692,-92.262,-176.669,11.618,149.516
C09718=1119.584,408.939,-92.301,-176.669,11.623,149.517
C09719=1119.580,409.186,-92.340,-176.668,11.628,149.518
C09720=1119.576,409.434,-92.379,-176.667,11.633,149.519
C09721=1119.574,409.681,-92.418,-176.666,11.638,149.520
C09722=1119.569,409.927,-92.456,-176.665,11.642,149.521
C09723=1119.566,410.174,-92.496,-176.665,11.647,149.522
C09724=1119.562,410.421,-92.535,-176.663,11.653,149.523
C09725=1119.559,410.668,-92.574,-176.663,11.658,149.524
C09726=1119.556,410.914,-92.613,-176.662,11.662,149.526
C09727=1119.552,411.161,-92.652,-176.661,11.668,149.527
C09728=1119.548,411.408,-92.691,-176.661,11.673,149.528
C09729=1119.544,411.656,-92.730,-176.660,11.677,149.529
C09730=1119.541,411.903,-92.769,-176.659,11.683,149.530
C09731=1119.537,412.150,-92.808,-176.659,11.688,149.531
C09732=1119.534,412.397,-92.848,-176.657,11.694,149.532
C09733=1119.531,412.643,-92.886,-176.657,11.699,149.534
C09734=1119.527,412.890,-92.926,-176.656,11.704,149.535
C09735=1119.523,413.137,-92.964,-176.656,11.709,149.536
C09736=1119.519,413.384,-93.004,-176.655,11.715,149.538
C09737=1119.516,413.631,-93.043,-176.654,11.720,149.539
C09738=1119.513,413.878,-93.083,-176.654,11.726,149.540
C09739=1119.510,414.124,-93.122,-176.653,11.731,149.541
C09740=1119.508,414.372,-93.161,-176.653,11.737,149.543
C09741=1119.506,414.619,-93.199,-176.652,11.742,149.544
C09742=1119.505,414.865,-93.239,-176.652,11.748,149.545
C09743=1119.505,415.112,-93.277,-176.652,11.753,149.547
C09744=1119.505,415.359,-93.316,-176.651,11.759,149.548
C09745=1119.505,415.606,-93.355,-176.651,11.764,149.549
C09746=1119.506,415.818,-93.388,-176.651,11.769,149.551
C09747=1119.508,416.029,-93.421,-176.650,11.774,149.552
C09748=1119.509,416.241,-93.454,-176.650,11.779,149.553
C09749=1119.512,416.452,-93.487,-176.650,11.784,149.554
C09750=1119.514,416.664,-93.520,-176.649,11.789,149.556
C09751=1119.517,416.875,-93.553,-176.649,11.794,149.557
C09752=1119.520,417.088,-93.585,-176.649,11.799,149.558
C09753=1119.523,417.299,-93.618,-176.648,11.804,149.559
C09754=1119.104,417.299,-93.681,-176.641,11.809,149.558
C09755=1119.101,417.086,-93.648,-176.641,11.803,149.557
C09756=1119.098,416.875,-93.615,-176.641,11.798,149.556
C09757=1119.094,416.663,-93.582,-176.642,11.794,149.555
C09758=1119.092,416.452,-93.550,-176.642,11.788,149.554
C09759=1119.090,416.240,-93.516,-176.642,11.783,149.552
C09760=1119.089,416.029,-93.484,-176.643,11.779,149.551
C09761=1119.087,415.818,-93.450,-176.643,11.774,149.550
C09762=1119.086,415.606,-93.417,-176.644,11.769,149.549
C09763=1119.086,415.359,-93.378,-176.644,11.763,149.547
C09764=1119.086,415.112,-93.339,-176.644,11.757,149.546
C09765=1119.086,414.865,-93.301,-176.645,11.752,149.545
C09766=1119.087,414.618,-93.262,-176.645,11.747,149.543
C09767=1119.088,414.371,-93.223,-176.646,11.741,149.542
C09768=1119.091,414.125,-93.184,-176.647,11.735,149.541
C09769=1119.093,413.877,-93.145,-176.647,11.730,149.539
C09770=1119.097,413.630,-93.106,-176.648,11.724,149.538
C09771=1119.100,413.384,-93.066,-176.648,11.719,149.537
C09772=1119.104,413.137,-93.027,-176.649,11.713,149.536
C09773=1119.108,412.890,-92.988,-176.650,11.708,149.534
C09774=1119.111,412.643,-92.949,-176.651,11.703,149.533
C09775=1119.115,412.396,-92.909,-176.651,11.697,149.532
C09776=1119.118,412.149,-92.871,-176.652,11.692,149.531
C09777=1119.121,411.902,-92.832,-176.653,11.687,149.530
C09778=1119.125,411.655,-92.792,-176.654,11.681,149.528
C09779=1119.129,411.408,-92.753,-176.654,11.676,149.527
C09780=1119.132,411.161,-92.714,-176.655,11.671,149.526
C09781=1119.136,410.914,-92.675,-176.656,11.666,149.525
C09782=1119.140,410.668,-92.636,-176.657,11.661,149.524
C09783=1119.143,410.421,-92.597,-176.658,11.656,149.523
C09784=1119.147,410.174,-92.558,-176.659,11.651,149.522
C09785=1119.150,409.927,-92.518,-176.660,11.646,149.521
C09786=1119.154,409.680,-92.480,-176.660,11.641,149.519
C09787=1119.158,409.433,-92.441,-176.661,11.636,149.518
C09788=1119.161,409.186,-92.402,-176.663,11.631,149.517
C09789=1119.164,408.939,-92.363,-176.663,11.626,149.516
C09790=1119.168,408.692,-92.324,-176.664,11.622,149.515
C09791=1119.171,408.445,-92.284,-176.665,11.617,149.514
C09792=1119.176,408.198,-92.246,-176.666,11.612,149.513
C09793=1119.179,407.952,-92.207,-176.667,11.607,149.512
C09794=1119.182,407.705,-92.168,-176.668,11.603,149.511
C09795=1119.186,407.458,-92.129,-176.669,11.599,149.511
C09796=1119.190,407.211,-92.090,-176.670,11.594,149.510
C09797=1119.193,406.964,-92.052,-176.671,11.590,149.509
C09798=1119.197,406.717,-92.013,-176.673,11.584,149.508
C09799=1119.201,406.470,-91.974,-176.673,11.580,149.507
C09800=1119.204,406.224,-91.935,-176.674,11.576,149.506
C09801=1119.208,405.976,-91.896,-176.676,11.571,149.505
C09802=1119.211,405.729,-91.857,-176.677,11.567,149.504
C09803=1119.215,405.482,-91.818,-176.678,11.563,149.503
C09804=1119.218,405.235,-91.780,-176.679,11.558,149.503
C09805=1119.222,404.989,-91.741,-176.680,11.554,149.502
C09806=1119.226,404.742,-91.702,-176.681,11.550,149.501
C09807=1119.229,404.495,-91.664,-176.683,11.546,149.500
C09808=1119.233,404.248,-91.625,-176.684,11.541,149.499
C09809=1119.237,404.000,-91.586,-176.685,11.537,149.498
C09810=1119.239,403.753,-91.547,-176.686,11.533,149.498
C09811=1119.243,403.542,-91.514,-176.687,11.530,149.497
C09812=1119.246,403.330,-91.481,-176.689,11.526,149.496
C09813=1119.249,403.118,-91.448,-176.689,11.523,149.496
C09814=1119.252,402.906,-91.414,-176.690,11.519,149.495
C09815=1119.256,402.694,-91.382,-176.692,11.515,149.495
C09816=1119.258,402.483,-91.349,-176.693,11.512,149.494
C09817=1119.261,402.271,-91.316,-176.694,11.509,149.493
C09818=1119.264,402.059,-91.282,-176.695,11.505,149.493
C09819=1119.269,401.812,-91.244,-176.697,11.501,149.492
C09820=1119.272,401.566,-91.206,-176.697,11.498,149.491
C09821=1119.276,401.318,-91.167,-176.699,11.494,149.491
C09822=1119.279,401.071,-91.128,-176.700,11.490,149.490
C09823=1119.283,400.825,-91.090,-176.702,11.486,149.490
C09824=1119.287,400.578,-91.051,-176.703,11.482,149.489
C09825=1119.290,400.330,-91.013,-176.704,11.479,149.488
C09826=1119.293,400.083,-90.974,-176.706,11.475,149.488
C09827=1119.297,399.837,-90.936,-176.708,11.471,149.487
C09828=1119.301,399.590,-90.897,-176.709,11.468,149.486
C09829=1119.304,399.343,-90.859,-176.710,11.464,149.486
C09830=1119.308,399.095,-90.820,-176.712,11.460,149.485
C09831=1119.312,398.849,-90.782,-176.714,11.457,149.485
C09832=1119.315,398.602,-90.744,-176.715,11.454,149.484
C09833=1119.319,398.354,-90.705,-176.717,11.450,149.484
C09834=1119.323,398.108,-90.667,-176.718,11.447,149.483
C09835=1119.327,397.860,-90.628,-176.719,11.443,149.483
C09836=1119.330,397.613,-90.590,-176.721,11.439,149.482
C09837=1119.334,397.366,-90.551,-176.722,11.436,149.482
C09838=1119.337,397.120,-90.514,-176.724,11.433,149.481
C09839=1119.341,396.872,-90.475,-176.725,11.430,149.481
C09840=1119.344,396.625,-90.436,-176.727,11.426,149.480
C09841=1119.348,396.379,-90.399,-176.729,11.422,149.480
C09842=1119.352,396.131,-90.360,-176.730,11.419,149.479
C09843=1119.355,395.884,-90.322,-176.732,11.416,149.479
C09844=1119.359,395.638,-90.283,-176.734,11.413,149.479
C09845=1119.362,395.390,-90.245,-176.736,11.409,149.478
C09846=1119.366,395.143,-90.207,-176.737,11.407,149.478
C09847=1119.370,394.896,-90.169,-176.739,11.403,149.477
C09848=1119.374,394.649,-90.131,-176.741,11.401,149.477
C09849=1119.378,394.403,-90.093,-176.742,11.398,149.477
C09850=1119.381,394.155,-90.055,-176.744,11.394,149.476
C09851=1119.385,393.908,-90.016,-176.745,11.391,149.476
C09852=1119.388,393.661,-89.978,-176.747,11.388,149.475
C09853=1119.392,393.414,-89.940,-176.749,11.385,149.475
C09854=1119.396,393.166,-89.902,-176.750,11.383,149.475
C09855=1119.399,392.920,-89.864,-176.753,11.379,149.474
C09856=1119.403,392.673,-89.825,-176.754,11.377,149.474
C09857=1119.407,392.426,-89.788,-176.757,11.373,149.474
C09858=1119.411,392.179,-89.749,-176.758,11.371,149.474
C09859=1119.414,391.932,-89.711,-176.759,11.368,149.473
C09860=1119.418,391.685,-89.674,-176.762,11.365,149.473
C09861=1119.422,391.437,-89.635,-176.763,11.362,149.473
C09862=1119.425,391.191,-89.597,-176.765,11.360,149.473
C09863=1119.429,390.944,-89.560,-176.767,11.357,149.472
C09864=1119.432,390.696,-89.522,-176.769,11.354,149.472
C09865=1119.436,390.449,-89.483,-176.771,11.351,149.472
C09866=1119.439,390.202,-89.445,-176.773,11.349,149.472
C09867=1119.443,389.990,-89.413,-176.775,11.347,149.472
C09868=1119.445,389.778,-89.380,-176.776,11.344,149.471
C09869=1119.449,389.567,-89.348,-176.778,11.341,149.471
C09870=1119.452,389.355,-89.316,-176.779,11.340,149.471
C09871=1119.455,389.143,-89.283,-176.781,11.338,149.471
C09872=1119.459,388.931,-89.250,-176.783,11.335,149.471
C09873=1119.462,388.719,-89.218,-176.785,11.333,149.471
C09874=1119.465,388.507,-89.185,-176.786,11.331,149.471
C09875=1119.469,388.260,-89.148,-176.788,11.329,149.470
C09876=1119.472,388.012,-89.110,-176.790,11.325,149.470
C09877=1119.476,387.766,-89.072,-176.792,11.323,149.470
C09878=1119.480,387.518,-89.034,-176.794,11.321,149.470
C09879=1119.483,387.271,-88.996,-176.796,11.319,149.470
C09880=1119.487,387.024,-88.958,-176.798,11.316,149.470
C09881=1119.490,386.777,-88.920,-176.800,11.314,149.470
C09882=1119.494,386.530,-88.884,-176.802,11.312,149.469
C09883=1119.498,386.282,-88.845,-176.805,11.309,149.469
C09884=1119.502,386.036,-88.807,-176.806,11.306,149.469
C09885=1119.505,385.789,-88.770,-176.808,11.304,149.469
C09886=1119.509,385.542,-88.732,-176.811,11.302,149.469
C09887=1119.512,385.295,-88.694,-176.812,11.300,149.469
C09888=1119.517,385.047,-88.657,-176.815,11.298,149.469
C09889=1119.520,384.800,-88.619,-176.817,11.295,149.469
C09890=1119.524,384.553,-88.581,-176.819,11.293,149.469
C09891=1119.527,384.306,-88.543,-176.821,11.291,149.469
C09892=1119.531,384.059,-88.506,-176.823,11.289,149.469
C09893=1119.534,383.812,-88.468,-176.825,11.286,149.469
C09894=1119.538,383.565,-88.431,-176.827,11.284,149.469
C09895=1119.542,383.317,-88.393,-176.829,11.282,149.469
C09896=1119.546,383.070,-88.355,-176.832,11.280,149.469
C09897=1119.550,382.824,-88.318,-176.836,11.277,149.469
C09898=1119.553,382.576,-88.281,-176.839,11.274,149.469
C09899=1119.557,382.329,-88.243,-176.842,11.272,149.469
C09900=1119.560,382.082,-88.205,-176.845,11.269,149.469
C09901=1119.564,381.835,-88.168,-176.848,11.267,149.470
C09902=1119.568,381.588,-88.130,-176.850,11.265,149.470
C09903=1119.572,381.340,-88.093,-176.854,11.262,149.470
C09904=1119.575,381.094,-88.056,-176.856,11.259,149.470
C09905=1119.579,380.846,-88.017,-176.860,11.257,149.470
C09906=1119.583,380.599,-87.980,-176.863,11.254,149.470
C09907=1119.587,380.352,-87.942,-176.866,11.251,149.470
C09908=1119.591,380.105,-87.906,-176.869,11.249,149.470
C09909=1119.594,379.858,-87.868,-176.872,11.246,149.470
C09910=1119.598,379.610,-87.831,-176.875,11.244,149.471
C09911=1119.602,379.364,-87.793,-176.878,11.242,149.471
C09912=1119.605,379.116,-87.756,-176.881,11.239,149.471
C09913=1119.609,378.868,-87.719,-176.884,11.236,149.471
C09914=1119.613,378.622,-87.682,-176.887,11.234,149.471
C09915=1119.617,378.374,-87.644,-176.890,11.231,149.471
C09916=1119.620,378.127,-87.607,-176.894,11.229,149.471
C09917=1119.625,377.880,-87.570,-176.896,11.227,149.472
C09918=1119.627,377.633,-87.533,-176.899,11.224,149.472
C09919=1119.631,377.386,-87.496,-176.903,11.222,149.472
C09920=1119.635,377.139,-87.459,-176.906,11.219,149.472
C09921=1119.639,376.891,-87.422,-176.909,11.217,149.472
C09922=1119.642,376.644,-87.384,-176.912,11.214,149.472
C09923=1119.645,376.432,-87.352,-176.915,11.212,149.473
C09924=1119.650,376.220,-87.321,-176.917,11.210,149.473
C09925=1119.652,376.008,-87.289,-176.920,11.208,149.473
C09926=1119.655,375.796,-87.257,-176.923,11.206,149.473
C09927=1119.659,375.584,-87.225,-176.925,11.204,149.473
C09928=1119.662,375.372,-87.193,-176.928,11.201,149.473
C09929=1119.665,375.160,-87.161,-176.931,11.200,149.473
C09930=1119.669,374.948,-87.130,-176.934,11.198,149.474
C09931=1119.672,374.701,-87.092,-176.936,11.195,149.474
C09932=1119.676,374.453,-87.055,-176.940,11.193,149.474
C09933=1119.680,374.206,-87.019,-176.943,11.190,149.474
C09934=1119.683,373.958,-86.981,-176.946,11.188,149.474
C09935=1119.687,373.711,-86.945,-176.950,11.185,149.475
C09936=1119.691,373.464,-86.908,-176.953,11.183,149.475
C09937=1119.695,373.218,-86.871,-176.956,11.181,149.475
C09938=1119.698,372.970,-86.833,-176.959,11.179,149.475
C09939=1119.702,372.723,-86.797,-176.962,11.176,149.475
C09940=1119.706,372.476,-86.760,-176.965,11.174,149.476
C09941=1119.710,372.228,-86.723,-176.969,11.171,149.476
C09942=1119.713,371.981,-86.686,-176.972,11.169,149.476
C09943=1119.717,371.734,-86.650,-176.975,11.166,149.476
C09944=1119.721,371.487,-86.613,-176.979,11.164,149.476
C09945=1119.725,371.239,-86.576,-176.981,11.162,149.477
C09946=1119.729,370.992,-86.539,-176.985,11.159,149.477
C09947=1119.732,370.745,-86.503,-176.988,11.157,149.477
C09948=1119.736,370.497,-86.466,-176.991,11.155,149.477
C09949=1119.740,370.250,-86.429,-176.995,11.152,149.477
C09950=1119.743,370.003,-86.393,-176.998,11.150,149.478
C09951=1119.747,369.756,-86.356,-177.001,11.147,149.478
C09952=1119.751,369.508,-86.319,-177.004,11.145,149.478
C09953=1119.754,369.261,-86.283,-177.008,11.142,149.478
C09954=1119.758,369.014,-86.246,-177.010,11.140,149.479
C09955=1119.763,368.766,-86.209,-177.014,11.138,149.479
C09956=1119.766,368.519,-86.173,-177.017,11.136,149.479
C09957=1119.770,368.272,-86.136,-177.021,11.133,149.479
C09958=1119.774,368.025,-86.099,-177.024,11.131,149.480
C09959=1119.777,367.777,-86.063,-177.027,11.128,149.480
C09960=1119.781,367.530,-86.027,-177.031,11.126,149.480
C09961=1119.785,367.283,-85.990,-177.034,11.123,149.480
C09962=1119.789,367.036,-85.953,-177.037,11.121,149.480
C09963=1119.792,366.788,-85.918,-177.041,11.119,149.481
C09964=1119.796,366.541,-85.881,-177.044,11.116,149.481
C09965=1119.801,366.294,-85.844,-177.048,11.114,149.481
C09966=1119.804,366.047,-85.808,-177.050,11.112,149.481
C09967=1119.808,365.799,-85.772,-177.054,11.110,149.482
C09968=1119.811,365.551,-85.735,-177.057,11.107,149.482
C09969=1119.815,365.304,-85.698,-177.060,11.105,149.482
C09970=1119.819,365.057,-85.663,-177.063,11.102,149.482
C09971=1119.823,364.810,-85.626,-177.067,11.100,149.483
C09972=1119.827,364.562,-85.590,-177.070,11.098,149.483
C09973=1119.831,364.315,-85.554,-177.074,11.095,149.483
C09974=1119.834,364.068,-85.517,-177.077,11.093,149.483
C09975=1119.838,363.820,-85.481,-177.080,11.090,149.484
C09976=1119.842,363.573,-85.445,-177.084,11.088,149.484
C09977=1119.845,363.326,-85.409,-177.087,11.086,149.484
C09978=1119.850,363.079,-85.372,-177.091,11.083,149.484
C09979=1119.853,362.866,-85.341,-177.093,11.081,149.485
C09980=1119.856,362.654,-85.310,-177.097,11.079,149.485
C09981=1119.859,362.442,-85.280,-177.099,11.077,149.485
C09982=1119.862,362.230,-85.249,-177.102,11.076,149.485
C09983=1119.865,362.017,-85.217,-177.105,11.073,149.485
C09984=1119.869,361.805,-85.186,-177.108,11.071,149.486
C09985=1119.873,361.593,-85.156,-177.111,11.069,149.486
C09986=1119.875,361.381,-85.125,-177.114,11.067,149.486
C09987=1119.879,361.133,-85.089,-177.117,11.065,149.486
C09988=1119.883,360.886,-85.052,-177.121,11.062,149.487
C09989=1119.887,360.638,-85.016,-177.124,11.060,149.487
C09990=1119.891,360.391,-84.981,-177.127,11.057,149.487
C09991=1119.894,360.144,-84.945,-177.130,11.055,149.487
C09992=1119.898,359.897,-84.909,-177.134,11.053,149.488
C09993=1119.902,359.649,-84.873,-177.137,11.050,149.488
C09994=1119.905,359.402,-84.837,-177.141,11.048,149.488
C09995=1119.909,359.154,-84.801,-177.144,11.045,149.488
C09996=1119.914,358.906,-84.765,-177.147,11.043,149.489
//INST
///DATE 2021/06/15 17:28
///ATTR SC,RW,RJ
////FRAME ROBOT
///GROUP1 RB1
NOP
MOVL C00000 V=800.0 PL=0
MOVL C00001 V=800.0 PL=0
MOVL C00002 V=800.0 PL=0
MOVL C00003 V=800.0 PL=0
MOVL C00004 V=800.0 PL=0
MOVL C00005 V=800.0 PL=0
MOVL C00006 V=800.0 PL=0
MOVL C00007 V=800.0 PL=0
MOVL C00008 V=800.0 PL=0
MOVL C00009 V=800.0 PL=0
MOVL C00010 V=800.0 PL=0
MOVL C00011 V=800.0 PL=0
MOVL C00012 V=800.0 PL=0
MOVL C00013 V=800.0 PL=0
MOVL C00014 V=800.0 PL=0
MOVL C00015 V=800.0 PL=0
MOVL C00016 V=800.0 PL=0
MOVL C00017 V=800.0 PL=0
MOVL C00018 V=800.0 PL=0
MOVL C00019 V=800.0 PL=0
MOVL C00020 V=800.0 PL=0
MOVL C00021 V=800.0 PL=0
MOVL C00022 V=800.0 PL=0
MOVL C00023 V=800.0 PL=0
MOVL C00024 V=800.0 PL=0
MOVL C00025 V=800.0 PL=0
MOVL C00026 V=800.0 PL=0
MOVL C00027 V=800.0 PL=0
MOVL C00028 V=800.0 PL=0
MOVL C00029 V=800.0 PL=0
MOVL C00030 V=800.0 PL=0
MOVL C00031 V=800.0 PL=0
MOVL C00032 V=800.0 PL=0
MOVL C00033 V=800.0 PL=0
MOVL C00034 V=800.0 PL=0
MOVL C00035 V=800.0 PL=0
MOVL C00036 V=800.0 PL=0
MOVL C00037 V=800.0 PL=0
MOVL C00038 V=800.0 PL=0
MOVL C00039 V=800.0 PL=0
MOVL C00040 V=800.0 PL=0
MOVL C00041 V=800.0 PL=0
MOVL C00042 V=800.0 PL=0
MOVL C00043 V=800.0 PL=0
MOVL C00044 V=800.0 PL=0
MOVL C00045 V=800.0 PL=0
MOVL C00046 V=800.0 PL=0
MOVL C00047 V=800.0 PL=0
MOVL C00048 V=800.0 PL=0
MOVL C00049 V=800.0 PL=0
MOVL C00050 V=800.0 PL=0
MOVL C00051 V=800.0 PL=0
MOVL C00052 V=800.0 PL=0
MOVL C00053 V=800.0 PL=0
MOVL C00054 V=800.0 PL=0
MOVL C00055 V=800.0 PL=0
MOVL C00056 V=800.0 PL=0
MOVL C00057 V=800.0 PL=0
MOVL C00058 V=800.0 PL=0
MOVL C00059 V=800.0 PL=0
MOVL C00060 V=800.0 PL=0
MOVL C00061 V=800.0 PL=0
MOVL C00062 V=800.0 PL=0
MOVL C00063 V=800.0 PL=0
MOVL C00064 V=800.0 PL=0
MOVL C00065 V=800.0 PL=0
MOVL C00066 V=800.0 PL=0
MOVL C00067 V=800.0 PL=0
MOVL C00068 V=800.0 PL=0
MOVL C00069 V=800.0 PL=0
MOVL C00070 V=800.0 PL=0
MOVL C00071 V=800.0 PL=0
MOVL C00072 V=800.0 PL=0
MOVL C00073 V=800.0 PL=0
MOVL C00074 V=800.0 PL=0
MOVL C00075 V=800.0 PL=0
MOVL C00076 V=800.0 PL=0
MOVL C00077 V=800.0 PL=0
MOVL C00078 V=800.0 PL=0
MOVL C00079 V=800.0 PL=0
MOVL C00080 V=800.0 PL=0
MOVL C00081 V=800.0 PL=0
MOVL C00082 V=800.0 PL=0
MOVL C00083 V=800.0 PL=0
MOVL C00084 V=800.0 PL=0
MOVL C00085 V=800.0 PL=0
MOVL C00086 V=800.0 PL=0
MOVL C00087 V=800.0 PL=0
MOVL C00088 V=800.0 PL=0
MOVL C00089 V=800.0 PL=0
MOVL C00090 V=800.0 PL=0
MOVL C00091 V=800.0 PL=0
MOVL C00092 V=800.0 PL=0
MOVL C00093 V=800.0 PL=0
MOVL C00094 V=800.0 PL=0
MOVL C00095 V=800.0 PL=0
MOVL C00096 V=800.0 PL=0
MOVL C00097 V=800.0 PL=0
MOVL C00098 V=800.0 PL=0
MOVL C00099 V=800.0 PL=0
MOVL C00100 V=800.0 PL=0
MOVL C00101 V=800.0 PL=0
MOVL C00102 V=800.0 PL=0
MOVL C00103 V=800.0 PL=0
MOVL C00104 V=800.0 PL=0
MOVL C00105 V=800.0 PL=0
MOVL C00106 V=800.0 PL=0
MOVL C00107 V=800.0 PL=0
MOVL C00108 V=800.0 PL=0
MOVL C00109 V=800.0 PL=0
MOVL C00110 V=800.0 PL=0
MOVL C00111 V=800.0 PL=0
MOVL C00112 V=800.0 PL=0
MOVL C00113 V=800.0 PL=0
MOVL C00114 V=800.0 PL=0
MOVL C00115 V=800.0 PL=0
MOVL C00116 V=800.0 PL=0
MOVL C00117 V=800.0 PL=0
MOVL C00118 V=800.0 PL=0
MOVL C00119 V=800.0 PL=0
MOVL C00120 V=800.0 PL=0
MOVL C00121 V=800.0 PL=0
MOVL C00122 V=800.0 PL=0
MOVL C00123 V=800.0 PL=0
MOVL C00124 V=800.0 PL=0
MOVL C00125 V=800.0 PL=0
MOVL C00126 V=800.0 PL=0
MOVL C00127 V=800.0 PL=0
MOVL C00128 V=800.0 PL=0
MOVL C00129 V=800.0 PL=0
MOVL C00130 V=800.0 PL=0
MOVL C00131 V=800.0 PL=0
MOVL C00132 V=800.0 PL=0
MOVL C00133 V=800.0 PL=0
MOVL C00134 V=800.0 PL=0
MOVL C00135 V=800.0 PL=0
MOVL C00136 V=800.0 PL=0
MOVL C00137 V=800.0 PL=0
MOVL C00138 V=800.0 PL=0
MOVL C00139 V=800.0 PL=0
MOVL C00140 V=800.0 PL=0
MOVL C00141 V=800.0 PL=0
MOVL C00142 V=800.0 PL=0
MOVL C00143 V=800.0 PL=0
MOVL C00144 V=800.0 PL=0
MOVL C00145 V=800.0 PL=0
MOVL C00146 V=800.0 PL=0
MOVL C00147 V=800.0 PL=0
MOVL C00148 V=800.0 PL=0
MOVL C00149 V=800.0 PL=0
MOVL C00150 V=800.0 PL=0
MOVL C00151 V=800.0 PL=0
MOVL C00152 V=800.0 PL=0
MOVL C00153 V=800.0 PL=0
MOVL C00154 V=800.0 PL=0
MOVL C00155 V=800.0 PL=0
MOVL C00156 V=800.0 PL=0
MOVL C00157 V=800.0 PL=0
MOVL C00158 V=800.0 PL=0
MOVL C00159 V=800.0 PL=0
MOVL C00160 V=800.0 PL=0
MOVL C00161 V=800.0 PL=0
MOVL C00162 V=800.0 PL=0
MOVL C00163 V=800.0 PL=0
MOVL C00164 V=800.0 PL=0
MOVL C00165 V=800.0 PL=0
MOVL C00166 V=800.0 PL=0
MOVL C00167 V=800.0 PL=0
MOVL C00168 V=800.0 PL=0
MOVL C00169 V=800.0 PL=0
MOVL C00170 V=800.0 PL=0
MOVL C00171 V=800.0 PL=0
MOVL C00172 V=800.0 PL=0
MOVL C00173 V=800.0 PL=0
MOVL C00174 V=800.0 PL=0
MOVL C00175 V=800.0 PL=0
MOVL C00176 V=800.0 PL=0
MOVL C00177 V=800.0 PL=0
MOVL C00178 V=800.0 PL=0
MOVL C00179 V=800.0 PL=0
MOVL C00180 V=800.0 PL=0
MOVL C00181 V=800.0 PL=0
MOVL C00182 V=800.0 PL=0
MOVL C00183 V=800.0 PL=0
MOVL C00184 V=800.0 PL=0
MOVL C00185 V=800.0 PL=0
MOVL C00186 V=800.0 PL=0
MOVL C00187 V=800.0 PL=0
MOVL C00188 V=800.0 PL=0
MOVL C00189 V=800.0 PL=0
MOVL C00190 V=800.0 PL=0
MOVL C00191 V=800.0 PL=0
MOVL C00192 V=800.0 PL=0
MOVL C00193 V=800.0 PL=0
MOVL C00194 V=800.0 PL=0
MOVL C00195 V=800.0 PL=0
MOVL C00196 V=800.0 PL=0
MOVL C00197 V=800.0 PL=0
MOVL C00198 V=800.0 PL=0
MOVL C00199 V=800.0 PL=0
MOVL C00200 V=800.0 PL=0
MOVL C00201 V=800.0 PL=0
MOVL C00202 V=800.0 PL=0
MOVL C00203 V=800.0 PL=0
MOVL C00204 V=800.0 PL=0
MOVL C00205 V=800.0 PL=0
MOVL C00206 V=800.0 PL=0
MOVL C00207 V=800.0 PL=0
MOVL C00208 V=800.0 PL=0
MOVL C00209 V=800.0 PL=0
MOVL C00210 V=800.0 PL=0
MOVL C00211 V=800.0 PL=0
MOVL C00212 V=800.0 PL=0
MOVL C00213 V=800.0 PL=0
MOVL C00214 V=800.0 PL=0
MOVL C00215 V=800.0 PL=0
MOVL C00216 V=800.0 PL=0
MOVL C00217 V=800.0 PL=0
MOVL C00218 V=800.0 PL=0
MOVL C00219 V=800.0 PL=0
MOVL C00220 V=800.0 PL=0
MOVL C00221 V=800.0 PL=0
MOVL C00222 V=800.0 PL=0
MOVL C00223 V=800.0 PL=0
MOVL C00224 V=800.0 PL=0
MOVL C00225 V=800.0 PL=0
MOVL C00226 V=800.0 PL=0
MOVL C00227 V=800.0 PL=0
MOVL C00228 V=800.0 PL=0
MOVL C00229 V=800.0 PL=0
MOVL C00230 V=800.0 PL=0
MOVL C00231 V=800.0 PL=0
MOVL C00232 V=800.0 PL=0
MOVL C00233 V=800.0 PL=0
MOVL C00234 V=800.0 PL=0
MOVL C00235 V=800.0 PL=0
MOVL C00236 V=800.0 PL=0
MOVL C00237 V=800.0 PL=0
MOVL C00238 V=800.0 PL=0
MOVL C00239 V=800.0 PL=0
MOVL C00240 V=800.0 PL=0
MOVL C00241 V=800.0 PL=0
MOVL C00242 V=800.0 PL=0
MOVL C00243 V=800.0 PL=0
MOVL C00244 V=800.0 PL=0
MOVL C00245 V=800.0 PL=0
MOVL C00246 V=800.0 PL=0
MOVL C00247 V=800.0 PL=0
MOVL C00248 V=800.0 PL=0
MOVL C00249 V=800.0 PL=0
MOVL C00250 V=800.0 PL=0
MOVL C00251 V=800.0 PL=0
MOVL C00252 V=800.0 PL=0
MOVL C00253 V=800.0 PL=0
MOVL C00254 V=800.0 PL=0
MOVL C00255 V=800.0 PL=0
MOVL C00256 V=800.0 PL=0
MOVL C00257 V=800.0 PL=0
MOVL C00258 V=800.0 PL=0
MOVL C00259 V=800.0 PL=0
MOVL C00260 V=800.0 PL=0
MOVL C00261 V=800.0 PL=0
MOVL C00262 V=800.0 PL=0
MOVL C00263 V=800.0 PL=0
MOVL C00264 V=800.0 PL=0
MOVL C00265 V=800.0 PL=0
MOVL C00266 V=800.0 PL=0
MOVL C00267 V=800.0 PL=0
MOVL C00268 V=800.0 PL=0
MOVL C00269 V=800.0 PL=0
MOVL C00270 V=800.0 PL=0
MOVL C00271 V=800.0 PL=0
MOVL C00272 V=800.0 PL=0
MOVL C00273 V=800.0 PL=0
MOVL C00274 V=800.0 PL=0
MOVL C00275 V=800.0 PL=0
MOVL C00276 V=800.0 PL=0
MOVL C00277 V=800.0 PL=0
MOVL C00278 V=800.0 PL=0
MOVL C00279 V=800.0 PL=0
MOVL C00280 V=800.0 PL=0
MOVL C00281 V=800.0 PL=0
MOVL C00282 V=800.0 PL=0
MOVL C00283 V=800.0 PL=0
MOVL C00284 V=800.0 PL=0
MOVL C00285 V=800.0 PL=0
MOVL C00286 V=800.0 PL=0
MOVL C00287 V=800.0 PL=0
MOVL C00288 V=800.0 PL=0
MOVL C00289 V=800.0 PL=0
MOVL C00290 V=800.0 PL=0
MOVL C00291 V=800.0 PL=0
MOVL C00292 V=800.0 PL=0
MOVL C00293 V=800.0 PL=0
MOVL C00294 V=800.0 PL=0
MOVL C00295 V=800.0 PL=0
MOVL C00296 V=800.0 PL=0
MOVL C00297 V=800.0 PL=0
MOVL C00298 V=800.0 PL=0
MOVL C00299 V=800.0 PL=0
MOVL C00300 V=800.0 PL=0
MOVL C00301 V=800.0 PL=0
MOVL C00302 V=800.0 PL=0
MOVL C00303 V=800.0 PL=0
MOVL C00304 V=800.0 PL=0
MOVL C00305 V=800.0 PL=0
MOVL C00306 V=800.0 PL=0
MOVL C00307 V=800.0 PL=0
MOVL C00308 V=800.0 PL=0
MOVL C00309 V=800.0 PL=0
MOVL C00310 V=800.0 PL=0
MOVL C00311 V=800.0 PL=0
MOVL C00312 V=800.0 PL=0
MOVL C00313 V=800.0 PL=0
MOVL C00314 V=800.0 PL=0
MOVL C00315 V=800.0 PL=0
MOVL C00316 V=800.0 PL=0
MOVL C00317 V=800.0 PL=0
MOVL C00318 V=800.0 PL=0
MOVL C00319 V=800.0 PL=0
MOVL C00320 V=800.0 PL=0
MOVL C00321 V=800.0 PL=0
MOVL C00322 V=800.0 PL=0
MOVL C00323 V=800.0 PL=0
MOVL C00324 V=800.0 PL=0
MOVL C00325 V=800.0 PL=0
MOVL C00326 V=800.0 PL=0
MOVL C00327 V=800.0 PL=0
MOVL C00328 V=800.0 PL=0
MOVL C00329 V=800.0 PL=0
MOVL C00330 V=800.0 PL=0
MOVL C00331 V=800.0 PL=0
MOVL C00332 V=800.0 PL=0
MOVL C00333 V=800.0 PL=0
MOVL C00334 V=800.0 PL=0
MOVL C00335 V=800.0 PL=0
MOVL C00336 V=800.0 PL=0
MOVL C00337 V=800.0 PL=0
MOVL C00338 V=800.0 PL=0
MOVL C00339 V=800.0 PL=0
MOVL C00340 V=800.0 PL=0
MOVL C00341 V=800.0 PL=0
MOVL C00342 V=800.0 PL=0
MOVL C00343 V=800.0 PL=0
MOVL C00344 V=800.0 PL=0
MOVL C00345 V=800.0 PL=0
MOVL C00346 V=800.0 PL=0
MOVL C00347 V=800.0 PL=0
MOVL C00348 V=800.0 PL=0
MOVL C00349 V=800.0 PL=0
MOVL C00350 V=800.0 PL=0
MOVL C00351 V=800.0 PL=0
MOVL C00352 V=800.0 PL=0
MOVL C00353 V=800.0 PL=0
MOVL C00354 V=800.0 PL=0
MOVL C00355 V=800.0 PL=0
MOVL C00356 V=800.0 PL=0
MOVL C00357 V=800.0 PL=0
MOVL C00358 V=800.0 PL=0
MOVL C00359 V=800.0 PL=0
MOVL C00360 V=800.0 PL=0
MOVL C00361 V=800.0 PL=0
MOVL C00362 V=800.0 PL=0
MOVL C00363 V=800.0 PL=0
MOVL C00364 V=800.0 PL=0
MOVL C00365 V=800.0 PL=0
MOVL C00366 V=800.0 PL=0
MOVL C00367 V=800.0 PL=0
MOVL C00368 V=800.0 PL=0
MOVL C00369 V=800.0 PL=0
MOVL C00370 V=800.0 PL=0
MOVL C00371 V=800.0 PL=0
MOVL C00372 V=800.0 PL=0
MOVL C00373 V=800.0 PL=0
MOVL C00374 V=800.0 PL=0
MOVL C00375 V=800.0 PL=0
MOVL C00376 V=800.0 PL=0
MOVL C00377 V=800.0 PL=0
MOVL C00378 V=800.0 PL=0
MOVL C00379 V=800.0 PL=0
MOVL C00380 V=800.0 PL=0
MOVL C00381 V=800.0 PL=0
MOVL C00382 V=800.0 PL=0
MOVL C00383 V=800.0 PL=0
MOVL C00384 V=800.0 PL=0
MOVL C00385 V=800.0 PL=0
MOVL C00386 V=800.0 PL=0
MOVL C00387 V=800.0 PL=0
MOVL C00388 V=800.0 PL=0
MOVL C00389 V=800.0 PL=0
MOVL C00390 V=800.0 PL=0
MOVL C00391 V=800.0 PL=0
MOVL C00392 V=800.0 PL=0
MOVL C00393 V=800.0 PL=0
MOVL C00394 V=800.0 PL=0
MOVL C00395 V=800.0 PL=0
MOVL C00396 V=800.0 PL=0
MOVL C00397 V=800.0 PL=0
MOVL C00398 V=800.0 PL=0
MOVL C00399 V=800.0 PL=0
MOVL C00400 V=800.0 PL=0
MOVL C00401 V=800.0 PL=0
MOVL C00402 V=800.0 PL=0
MOVL C00403 V=800.0 PL=0
MOVL C00404 V=800.0 PL=0
MOVL C00405 V=800.0 PL=0
MOVL C00406 V=800.0 PL=0
MOVL C00407 V=800.0 PL=0
MOVL C00408 V=800.0 PL=0
MOVL C00409 V=800.0 PL=0
MOVL C00410 V=800.0 PL=0
MOVL C00411 V=800.0 PL=0
MOVL C00412 V=800.0 PL=0
MOVL C00413 V=800.0 PL=0
MOVL C00414 V=800.0 PL=0
MOVL C00415 V=800.0 PL=0
MOVL C00416 V=800.0 PL=0
MOVL C00417 V=800.0 PL=0
MOVL C00418 V=800.0 PL=0
MOVL C00419 V=800.0 PL=0
MOVL C00420 V=800.0 PL=0
MOVL C00421 V=800.0 PL=0
MOVL C00422 V=800.0 PL=0
MOVL C00423 V=800.0 PL=0
MOVL C00424 V=800.0 PL=0
MOVL C00425 V=800.0 PL=0
MOVL C00426 V=800.0 PL=0
MOVL C00427 V=800.0 PL=0
MOVL C00428 V=800.0 PL=0
MOVL C00429 V=800.0 PL=0
MOVL C00430 V=800.0 PL=0
MOVL C00431 V=800.0 PL=0
MOVL C00432 V=800.0 PL=0
MOVL C00433 V=800.0 PL=0
MOVL C00434 V=800.0 PL=0
MOVL C00435 V=800.0 PL=0
MOVL C00436 V=800.0 PL=0
MOVL C00437 V=800.0 PL=0
MOVL C00438 V=800.0 PL=0
MOVL C00439 V=800.0 PL=0
MOVL C00440 V=800.0 PL=0
MOVL C00441 V=800.0 PL=0
MOVL C00442 V=800.0 PL=0
MOVL C00443 V=800.0 PL=0
MOVL C00444 V=800.0 PL=0
MOVL C00445 V=800.0 PL=0
MOVL C00446 V=800.0 PL=0
MOVL C00447 V=800.0 PL=0
MOVL C00448 V=800.0 PL=0
MOVL C00449 V=800.0 PL=0
MOVL C00450 V=800.0 PL=0
MOVL C00451 V=800.0 PL=0
MOVL C00452 V=800.0 PL=0
MOVL C00453 V=800.0 PL=0
MOVL C00454 V=800.0 PL=0
MOVL C00455 V=800.0 PL=0
MOVL C00456 V=800.0 PL=0
MOVL C00457 V=800.0 PL=0
MOVL C00458 V=800.0 PL=0
MOVL C00459 V=800.0 PL=0
MOVL C00460 V=800.0 PL=0
MOVL C00461 V=800.0 PL=0
MOVL C00462 V=800.0 PL=0
MOVL C00463 V=800.0 PL=0
MOVL C00464 V=800.0 PL=0
MOVL C00465 V=800.0 PL=0
MOVL C00466 V=800.0 PL=0
MOVL C00467 V=800.0 PL=0
MOVL C00468 V=800.0 PL=0
MOVL C00469 V=800.0 PL=0
MOVL C00470 V=800.0 PL=0
MOVL C00471 V=800.0 PL=0
MOVL C00472 V=800.0 PL=0
MOVL C00473 V=800.0 PL=0
MOVL C00474 V=800.0 PL=0
MOVL C00475 V=800.0 PL=0
MOVL C00476 V=800.0 PL=0
MOVL C00477 V=800.0 PL=0
MOVL C00478 V=800.0 PL=0
MOVL C00479 V=800.0 PL=0
MOVL C00480 V=800.0 PL=0
MOVL C00481 V=800.0 PL=0
MOVL C00482 V=800.0 PL=0
MOVL C00483 V=800.0 PL=0
MOVL C00484 V=800.0 PL=0
MOVL C00485 V=800.0 PL=0
MOVL C00486 V=800.0 PL=0
MOVL C00487 V=800.0 PL=0
MOVL C00488 V=800.0 PL=0
MOVL C00489 V=800.0 PL=0
MOVL C00490 V=800.0 PL=0
MOVL C00491 V=800.0 PL=0
MOVL C00492 V=800.0 PL=0
MOVL C00493 V=800.0 PL=0
MOVL C00494 V=800.0 PL=0
MOVL C00495 V=800.0 PL=0
MOVL C00496 V=800.0 PL=0
MOVL C00497 V=800.0 PL=0
MOVL C00498 V=800.0 PL=0
MOVL C00499 V=800.0 PL=0
MOVL C00500 V=800.0 PL=0
MOVL C00501 V=800.0 PL=0
MOVL C00502 V=800.0 PL=0
MOVL C00503 V=800.0 PL=0
MOVL C00504 V=800.0 PL=0
MOVL C00505 V=800.0 PL=0
MOVL C00506 V=800.0 PL=0
MOVL C00507 V=800.0 PL=0
MOVL C00508 V=800.0 PL=0
MOVL C00509 V=800.0 PL=0
MOVL C00510 V=800.0 PL=0
MOVL C00511 V=800.0 PL=0
MOVL C00512 V=800.0 PL=0
MOVL C00513 V=800.0 PL=0
MOVL C00514 V=800.0 PL=0
MOVL C00515 V=800.0 PL=0
MOVL C00516 V=800.0 PL=0
MOVL C00517 V=800.0 PL=0
MOVL C00518 V=800.0 PL=0
MOVL C00519 V=800.0 PL=0
MOVL C00520 V=800.0 PL=0
MOVL C00521 V=800.0 PL=0
MOVL C00522 V=800.0 PL=0
MOVL C00523 V=800.0 PL=0
MOVL C00524 V=800.0 PL=0
MOVL C00525 V=800.0 PL=0
MOVL C00526 V=800.0 PL=0
MOVL C00527 V=800.0 PL=0
MOVL C00528 V=800.0 PL=0
MOVL C00529 V=800.0 PL=0
MOVL C00530 V=800.0 PL=0
MOVL C00531 V=800.0 PL=0
MOVL C00532 V=800.0 PL=0
MOVL C00533 V=800.0 PL=0
MOVL C00534 V=800.0 PL=0
MOVL C00535 V=800.0 PL=0
MOVL C00536 V=800.0 PL=0
MOVL C00537 V=800.0 PL=0
MOVL C00538 V=800.0 PL=0
MOVL C00539 V=800.0 PL=0
MOVL C00540 V=800.0 PL=0
MOVL C00541 V=800.0 PL=0
MOVL C00542 V=800.0 PL=0
MOVL C00543 V=800.0 PL=0
MOVL C00544 V=800.0 PL=0
MOVL C00545 V=800.0 PL=0
MOVL C00546 V=800.0 PL=0
MOVL C00547 V=800.0 PL=0
MOVL C00548 V=800.0 PL=0
MOVL C00549 V=800.0 PL=0
MOVL C00550 V=800.0 PL=0
MOVL C00551 V=800.0 PL=0
MOVL C00552 V=800.0 PL=0
MOVL C00553 V=800.0 PL=0
MOVL C00554 V=800.0 PL=0
MOVL C00555 V=800.0 PL=0
MOVL C00556 V=800.0 PL=0
MOVL C00557 V=800.0 PL=0
MOVL C00558 V=800.0 PL=0
MOVL C00559 V=800.0 PL=0
MOVL C00560 V=800.0 PL=0
MOVL C00561 V=800.0 PL=0
MOVL C00562 V=800.0 PL=0
MOVL C00563 V=800.0 PL=0
MOVL C00564 V=800.0 PL=0
MOVL C00565 V=800.0 PL=0
MOVL C00566 V=800.0 PL=0
MOVL C00567 V=800.0 PL=0
MOVL C00568 V=800.0 PL=0
MOVL C00569 V=800.0 PL=0
MOVL C00570 V=800.0 PL=0
MOVL C00571 V=800.0 PL=0
MOVL C00572 V=800.0 PL=0
MOVL C00573 V=800.0 PL=0
MOVL C00574 V=800.0 PL=0
MOVL C00575 V=800.0 PL=0
MOVL C00576 V=800.0 PL=0
MOVL C00577 V=800.0 PL=0
MOVL C00578 V=800.0 PL=0
MOVL C00579 V=800.0 PL=0
MOVL C00580 V=800.0 PL=0
MOVL C00581 V=800.0 PL=0
MOVL C00582 V=800.0 PL=0
MOVL C00583 V=800.0 PL=0
MOVL C00584 V=800.0 PL=0
MOVL C00585 V=800.0 PL=0
MOVL C00586 V=800.0 PL=0
MOVL C00587 V=800.0 PL=0
MOVL C00588 V=800.0 PL=0
MOVL C00589 V=800.0 PL=0
MOVL C00590 V=800.0 PL=0
MOVL C00591 V=800.0 PL=0
MOVL C00592 V=800.0 PL=0
MOVL C00593 V=800.0 PL=0
MOVL C00594 V=800.0 PL=0
MOVL C00595 V=800.0 PL=0
MOVL C00596 V=800.0 PL=0
MOVL C00597 V=800.0 PL=0
MOVL C00598 V=800.0 PL=0
MOVL C00599 V=800.0 PL=0
MOVL C00600 V=800.0 PL=0
MOVL C00601 V=800.0 PL=0
MOVL C00602 V=800.0 PL=0
MOVL C00603 V=800.0 PL=0
MOVL C00604 V=800.0 PL=0
MOVL C00605 V=800.0 PL=0
MOVL C00606 V=800.0 PL=0
MOVL C00607 V=800.0 PL=0
MOVL C00608 V=800.0 PL=0
MOVL C00609 V=800.0 PL=0
MOVL C00610 V=800.0 PL=0
MOVL C00611 V=800.0 PL=0
MOVL C00612 V=800.0 PL=0
MOVL C00613 V=800.0 PL=0
MOVL C00614 V=800.0 PL=0
MOVL C00615 V=800.0 PL=0
MOVL C00616 V=800.0 PL=0
MOVL C00617 V=800.0 PL=0
MOVL C00618 V=800.0 PL=0
MOVL C00619 V=800.0 PL=0
MOVL C00620 V=800.0 PL=0
MOVL C00621 V=800.0 PL=0
MOVL C00622 V=800.0 PL=0
MOVL C00623 V=800.0 PL=0
MOVL C00624 V=800.0 PL=0
MOVL C00625 V=800.0 PL=0
MOVL C00626 V=800.0 PL=0
MOVL C00627 V=800.0 PL=0
MOVL C00628 V=800.0 PL=0
MOVL C00629 V=800.0 PL=0
MOVL C00630 V=800.0 PL=0
MOVL C00631 V=800.0 PL=0
MOVL C00632 V=800.0 PL=0
MOVL C00633 V=800.0 PL=0
MOVL C00634 V=800.0 PL=0
MOVL C00635 V=800.0 PL=0
MOVL C00636 V=800.0 PL=0
MOVL C00637 V=800.0 PL=0
MOVL C00638 V=800.0 PL=0
MOVL C00639 V=800.0 PL=0
MOVL C00640 V=800.0 PL=0
MOVL C00641 V=800.0 PL=0
MOVL C00642 V=800.0 PL=0
MOVL C00643 V=800.0 PL=0
MOVL C00644 V=800.0 PL=0
MOVL C00645 V=800.0 PL=0
MOVL C00646 V=800.0 PL=0
MOVL C00647 V=800.0 PL=0
MOVL C00648 V=800.0 PL=0
MOVL C00649 V=800.0 PL=0
MOVL C00650 V=800.0 PL=0
MOVL C00651 V=800.0 PL=0
MOVL C00652 V=800.0 PL=0
MOVL C00653 V=800.0 PL=0
MOVL C00654 V=800.0 PL=0
MOVL C00655 V=800.0 PL=0
MOVL C00656 V=800.0 PL=0
MOVL C00657 V=800.0 PL=0
MOVL C00658 V=800.0 PL=0
MOVL C00659 V=800.0 PL=0
MOVL C00660 V=800.0 PL=0
MOVL C00661 V=800.0 PL=0
MOVL C00662 V=800.0 PL=0
MOVL C00663 V=800.0 PL=0
MOVL C00664 V=800.0 PL=0
MOVL C00665 V=800.0 PL=0
MOVL C00666 V=800.0 PL=0
MOVL C00667 V=800.0 PL=0
MOVL C00668 V=800.0 PL=0
MOVL C00669 V=800.0 PL=0
MOVL C00670 V=800.0 PL=0
MOVL C00671 V=800.0 PL=0
MOVL C00672 V=800.0 PL=0
MOVL C00673 V=800.0 PL=0
MOVL C00674 V=800.0 PL=0
MOVL C00675 V=800.0 PL=0
MOVL C00676 V=800.0 PL=0
MOVL C00677 V=800.0 PL=0
MOVL C00678 V=800.0 PL=0
MOVL C00679 V=800.0 PL=0
MOVL C00680 V=800.0 PL=0
MOVL C00681 V=800.0 PL=0
MOVL C00682 V=800.0 PL=0
MOVL C00683 V=800.0 PL=0
MOVL C00684 V=800.0 PL=0
MOVL C00685 V=800.0 PL=0
MOVL C00686 V=800.0 PL=0
MOVL C00687 V=800.0 PL=0
MOVL C00688 V=800.0 PL=0
MOVL C00689 V=800.0 PL=0
MOVL C00690 V=800.0 PL=0
MOVL C00691 V=800.0 PL=0
MOVL C00692 V=800.0 PL=0
MOVL C00693 V=800.0 PL=0
MOVL C00694 V=800.0 PL=0
MOVL C00695 V=800.0 PL=0
MOVL C00696 V=800.0 PL=0
MOVL C00697 V=800.0 PL=0
MOVL C00698 V=800.0 PL=0
MOVL C00699 V=800.0 PL=0
MOVL C00700 V=800.0 PL=0
MOVL C00701 V=800.0 PL=0
MOVL C00702 V=800.0 PL=0
MOVL C00703 V=800.0 PL=0
MOVL C00704 V=800.0 PL=0
MOVL C00705 V=800.0 PL=0
MOVL C00706 V=800.0 PL=0
MOVL C00707 V=800.0 PL=0
MOVL C00708 V=800.0 PL=0
MOVL C00709 V=800.0 PL=0
MOVL C00710 V=800.0 PL=0
MOVL C00711 V=800.0 PL=0
MOVL C00712 V=800.0 PL=0
MOVL C00713 V=800.0 PL=0
MOVL C00714 V=800.0 PL=0
MOVL C00715 V=800.0 PL=0
MOVL C00716 V=800.0 PL=0
MOVL C00717 V=800.0 PL=0
MOVL C00718 V=800.0 PL=0
MOVL C00719 V=800.0 PL=0
MOVL C00720 V=800.0 PL=0
MOVL C00721 V=800.0 PL=0
MOVL C00722 V=800.0 PL=0
MOVL C00723 V=800.0 PL=0
MOVL C00724 V=800.0 PL=0
MOVL C00725 V=800.0 PL=0
MOVL C00726 V=800.0 PL=0
MOVL C00727 V=800.0 PL=0
MOVL C00728 V=800.0 PL=0
MOVL C00729 V=800.0 PL=0
MOVL C00730 V=800.0 PL=0
MOVL C00731 V=800.0 PL=0
MOVL C00732 V=800.0 PL=0
MOVL C00733 V=800.0 PL=0
MOVL C00734 V=800.0 PL=0
MOVL C00735 V=800.0 PL=0
MOVL C00736 V=800.0 PL=0
MOVL C00737 V=800.0 PL=0
MOVL C00738 V=800.0 PL=0
MOVL C00739 V=800.0 PL=0
MOVL C00740 V=800.0 PL=0
MOVL C00741 V=800.0 PL=0
MOVL C00742 V=800.0 PL=0
MOVL C00743 V=800.0 PL=0
MOVL C00744 V=800.0 PL=0
MOVL C00745 V=800.0 PL=0
MOVL C00746 V=800.0 PL=0
MOVL C00747 V=800.0 PL=0
MOVL C00748 V=800.0 PL=0
MOVL C00749 V=800.0 PL=0
MOVL C00750 V=800.0 PL=0
MOVL C00751 V=800.0 PL=0
MOVL C00752 V=800.0 PL=0
MOVL C00753 V=800.0 PL=0
MOVL C00754 V=800.0 PL=0
MOVL C00755 V=800.0 PL=0
MOVL C00756 V=800.0 PL=0
MOVL C00757 V=800.0 PL=0
MOVL C00758 V=800.0 PL=0
MOVL C00759 V=800.0 PL=0
MOVL C00760 V=800.0 PL=0
MOVL C00761 V=800.0 PL=0
MOVL C00762 V=800.0 PL=0
MOVL C00763 V=800.0 PL=0
MOVL C00764 V=800.0 PL=0
MOVL C00765 V=800.0 PL=0
MOVL C00766 V=800.0 PL=0
MOVL C00767 V=800.0 PL=0
MOVL C00768 V=800.0 PL=0
MOVL C00769 V=800.0 PL=0
MOVL C00770 V=800.0 PL=0
MOVL C00771 V=800.0 PL=0
MOVL C00772 V=800.0 PL=0
MOVL C00773 V=800.0 PL=0
MOVL C00774 V=800.0 PL=0
MOVL C00775 V=800.0 PL=0
MOVL C00776 V=800.0 PL=0
MOVL C00777 V=800.0 PL=0
MOVL C00778 V=800.0 PL=0
MOVL C00779 V=800.0 PL=0
MOVL C00780 V=800.0 PL=0
MOVL C00781 V=800.0 PL=0
MOVL C00782 V=800.0 PL=0
MOVL C00783 V=800.0 PL=0
MOVL C00784 V=800.0 PL=0
MOVL C00785 V=800.0 PL=0
MOVL C00786 V=800.0 PL=0
MOVL C00787 V=800.0 PL=0
MOVL C00788 V=800.0 PL=0
MOVL C00789 V=800.0 PL=0
MOVL C00790 V=800.0 PL=0
MOVL C00791 V=800.0 PL=0
MOVL C00792 V=800.0 PL=0
MOVL C00793 V=800.0 PL=0
MOVL C00794 V=800.0 PL=0
MOVL C00795 V=800.0 PL=0
MOVL C00796 V=800.0 PL=0
MOVL C00797 V=800.0 PL=0
MOVL C00798 V=800.0 PL=0
MOVL C00799 V=800.0 PL=0
MOVL C00800 V=800.0 PL=0
MOVL C00801 V=800.0 PL=0
MOVL C00802 V=800.0 PL=0
MOVL C00803 V=800.0 PL=0
MOVL C00804 V=800.0 PL=0
MOVL C00805 V=800.0 PL=0
MOVL C00806 V=800.0 PL=0
MOVL C00807 V=800.0 PL=0
MOVL C00808 V=800.0 PL=0
MOVL C00809 V=800.0 PL=0
MOVL C00810 V=800.0 PL=0
MOVL C00811 V=800.0 PL=0
MOVL C00812 V=800.0 PL=0
MOVL C00813 V=800.0 PL=0
MOVL C00814 V=800.0 PL=0
MOVL C00815 V=800.0 PL=0
MOVL C00816 V=800.0 PL=0
MOVL C00817 V=800.0 PL=0
MOVL C00818 V=800.0 PL=0
MOVL C00819 V=800.0 PL=0
MOVL C00820 V=800.0 PL=0
MOVL C00821 V=800.0 PL=0
MOVL C00822 V=800.0 PL=0
MOVL C00823 V=800.0 PL=0
MOVL C00824 V=800.0 PL=0
MOVL C00825 V=800.0 PL=0
MOVL C00826 V=800.0 PL=0
MOVL C00827 V=800.0 PL=0
MOVL C00828 V=800.0 PL=0
MOVL C00829 V=800.0 PL=0
MOVL C00830 V=800.0 PL=0
MOVL C00831 V=800.0 PL=0
MOVL C00832 V=800.0 PL=0
MOVL C00833 V=800.0 PL=0
MOVL C00834 V=800.0 PL=0
MOVL C00835 V=800.0 PL=0
MOVL C00836 V=800.0 PL=0
MOVL C00837 V=800.0 PL=0
MOVL C00838 V=800.0 PL=0
MOVL C00839 V=800.0 PL=0
MOVL C00840 V=800.0 PL=0
MOVL C00841 V=800.0 PL=0
MOVL C00842 V=800.0 PL=0
MOVL C00843 V=800.0 PL=0
MOVL C00844 V=800.0 PL=0
MOVL C00845 V=800.0 PL=0
MOVL C00846 V=800.0 PL=0
MOVL C00847 V=800.0 PL=0
MOVL C00848 V=800.0 PL=0
MOVL C00849 V=800.0 PL=0
MOVL C00850 V=800.0 PL=0
MOVL C00851 V=800.0 PL=0
MOVL C00852 V=800.0 PL=0
MOVL C00853 V=800.0 PL=0
MOVL C00854 V=800.0 PL=0
MOVL C00855 V=800.0 PL=0
MOVL C00856 V=800.0 PL=0
MOVL C00857 V=800.0 PL=0
MOVL C00858 V=800.0 PL=0
MOVL C00859 V=800.0 PL=0
MOVL C00860 V=800.0 PL=0
MOVL C00861 V=800.0 PL=0
MOVL C00862 V=800.0 PL=0
MOVL C00863 V=800.0 PL=0
MOVL C00864 V=800.0 PL=0
MOVL C00865 V=800.0 PL=0
MOVL C00866 V=800.0 PL=0
MOVL C00867 V=800.0 PL=0
MOVL C00868 V=800.0 PL=0
MOVL C00869 V=800.0 PL=0
MOVL C00870 V=800.0 PL=0
MOVL C00871 V=800.0 PL=0
MOVL C00872 V=800.0 PL=0
MOVL C00873 V=800.0 PL=0
MOVL C00874 V=800.0 PL=0
MOVL C00875 V=800.0 PL=0
MOVL C00876 V=800.0 PL=0
MOVL C00877 V=800.0 PL=0
MOVL C00878 V=800.0 PL=0
MOVL C00879 V=800.0 PL=0
MOVL C00880 V=800.0 PL=0
MOVL C00881 V=800.0 PL=0
MOVL C00882 V=800.0 PL=0
MOVL C00883 V=800.0 PL=0
MOVL C00884 V=800.0 PL=0
MOVL C00885 V=800.0 PL=0
MOVL C00886 V=800.0 PL=0
MOVL C00887 V=800.0 PL=0
MOVL C00888 V=800.0 PL=0
MOVL C00889 V=800.0 PL=0
MOVL C00890 V=800.0 PL=0
MOVL C00891 V=800.0 PL=0
MOVL C00892 V=800.0 PL=0
MOVL C00893 V=800.0 PL=0
MOVL C00894 V=800.0 PL=0
MOVL C00895 V=800.0 PL=0
MOVL C00896 V=800.0 PL=0
MOVL C00897 V=800.0 PL=0
MOVL C00898 V=800.0 PL=0
MOVL C00899 V=800.0 PL=0
MOVL C00900 V=800.0 PL=0
MOVL C00901 V=800.0 PL=0
MOVL C00902 V=800.0 PL=0
MOVL C00903 V=800.0 PL=0
MOVL C00904 V=800.0 PL=0
MOVL C00905 V=800.0 PL=0
MOVL C00906 V=800.0 PL=0
MOVL C00907 V=800.0 PL=0
MOVL C00908 V=800.0 PL=0
MOVL C00909 V=800.0 PL=0
MOVL C00910 V=800.0 PL=0
MOVL C00911 V=800.0 PL=0
MOVL C00912 V=800.0 PL=0
MOVL C00913 V=800.0 PL=0
MOVL C00914 V=800.0 PL=0
MOVL C00915 V=800.0 PL=0
MOVL C00916 V=800.0 PL=0
MOVL C00917 V=800.0 PL=0
MOVL C00918 V=800.0 PL=0
MOVL C00919 V=800.0 PL=0
MOVL C00920 V=800.0 PL=0
MOVL C00921 V=800.0 PL=0
MOVL C00922 V=800.0 PL=0
MOVL C00923 V=800.0 PL=0
MOVL C00924 V=800.0 PL=0
MOVL C00925 V=800.0 PL=0
MOVL C00926 V=800.0 PL=0
MOVL C00927 V=800.0 PL=0
MOVL C00928 V=800.0 PL=0
MOVL C00929 V=800.0 PL=0
MOVL C00930 V=800.0 PL=0
MOVL C00931 V=800.0 PL=0
MOVL C00932 V=800.0 PL=0
MOVL C00933 V=800.0 PL=0
MOVL C00934 V=800.0 PL=0
MOVL C00935 V=800.0 PL=0
MOVL C00936 V=800.0 PL=0
MOVL C00937 V=800.0 PL=0
MOVL C00938 V=800.0 PL=0
MOVL C00939 V=800.0 PL=0
MOVL C00940 V=800.0 PL=0
MOVL C00941 V=800.0 PL=0
MOVL C00942 V=800.0 PL=0
MOVL C00943 V=800.0 PL=0
MOVL C00944 V=800.0 PL=0
MOVL C00945 V=800.0 PL=0
MOVL C00946 V=800.0 PL=0
MOVL C00947 V=800.0 PL=0
MOVL C00948 V=800.0 PL=0
MOVL C00949 V=800.0 PL=0
MOVL C00950 V=800.0 PL=0
MOVL C00951 V=800.0 PL=0
MOVL C00952 V=800.0 PL=0
MOVL C00953 V=800.0 PL=0
MOVL C00954 V=800.0 PL=0
MOVL C00955 V=800.0 PL=0
MOVL C00956 V=800.0 PL=0
MOVL C00957 V=800.0 PL=0
MOVL C00958 V=800.0 PL=0
MOVL C00959 V=800.0 PL=0
MOVL C00960 V=800.0 PL=0
MOVL C00961 V=800.0 PL=0
MOVL C00962 V=800.0 PL=0
MOVL C00963 V=800.0 PL=0
MOVL C00964 V=800.0 PL=0
MOVL C00965 V=800.0 PL=0
MOVL C00966 V=800.0 PL=0
MOVL C00967 V=800.0 PL=0
MOVL C00968 V=800.0 PL=0
MOVL C00969 V=800.0 PL=0
MOVL C00970 V=800.0 PL=0
MOVL C00971 V=800.0 PL=0
MOVL C00972 V=800.0 PL=0
MOVL C00973 V=800.0 PL=0
MOVL C00974 V=800.0 PL=0
MOVL C00975 V=800.0 PL=0
MOVL C00976 V=800.0 PL=0
MOVL C00977 V=800.0 PL=0
MOVL C00978 V=800.0 PL=0
MOVL C00979 V=800.0 PL=0
MOVL C00980 V=800.0 PL=0
MOVL C00981 V=800.0 PL=0
MOVL C00982 V=800.0 PL=0
MOVL C00983 V=800.0 PL=0
MOVL C00984 V=800.0 PL=0
MOVL C00985 V=800.0 PL=0
MOVL C00986 V=800.0 PL=0
MOVL C00987 V=800.0 PL=0
MOVL C00988 V=800.0 PL=0
MOVL C00989 V=800.0 PL=0
MOVL C00990 V=800.0 PL=0
MOVL C00991 V=800.0 PL=0
MOVL C00992 V=800.0 PL=0
MOVL C00993 V=800.0 PL=0
MOVL C00994 V=800.0 PL=0
MOVL C00995 V=800.0 PL=0
MOVL C00996 V=800.0 PL=0
MOVL C00997 V=800.0 PL=0
MOVL C00998 V=800.0 PL=0
MOVL C00999 V=800.0 PL=0
MOVL C01000 V=800.0 PL=0
MOVL C01001 V=800.0 PL=0
MOVL C01002 V=800.0 PL=0
MOVL C01003 V=800.0 PL=0
MOVL C01004 V=800.0 PL=0
MOVL C01005 V=800.0 PL=0
MOVL C01006 V=800.0 PL=0
MOVL C01007 V=800.0 PL=0
MOVL C01008 V=800.0 PL=0
MOVL C01009 V=800.0 PL=0
MOVL C01010 V=800.0 PL=0
MOVL C01011 V=800.0 PL=0
MOVL C01012 V=800.0 PL=0
MOVL C01013 V=800.0 PL=0
MOVL C01014 V=800.0 PL=0
MOVL C01015 V=800.0 PL=0
MOVL C01016 V=800.0 PL=0
MOVL C01017 V=800.0 PL=0
MOVL C01018 V=800.0 PL=0
MOVL C01019 V=800.0 PL=0
MOVL C01020 V=800.0 PL=0
MOVL C01021 V=800.0 PL=0
MOVL C01022 V=800.0 PL=0
MOVL C01023 V=800.0 PL=0
MOVL C01024 V=800.0 PL=0
MOVL C01025 V=800.0 PL=0
MOVL C01026 V=800.0 PL=0
MOVL C01027 V=800.0 PL=0
MOVL C01028 V=800.0 PL=0
MOVL C01029 V=800.0 PL=0
MOVL C01030 V=800.0 PL=0
MOVL C01031 V=800.0 PL=0
MOVL C01032 V=800.0 PL=0
MOVL C01033 V=800.0 PL=0
MOVL C01034 V=800.0 PL=0
MOVL C01035 V=800.0 PL=0
MOVL C01036 V=800.0 PL=0
MOVL C01037 V=800.0 PL=0
MOVL C01038 V=800.0 PL=0
MOVL C01039 V=800.0 PL=0
MOVL C01040 V=800.0 PL=0
MOVL C01041 V=800.0 PL=0
MOVL C01042 V=800.0 PL=0
MOVL C01043 V=800.0 PL=0
MOVL C01044 V=800.0 PL=0
MOVL C01045 V=800.0 PL=0
MOVL C01046 V=800.0 PL=0
MOVL C01047 V=800.0 PL=0
MOVL C01048 V=800.0 PL=0
MOVL C01049 V=800.0 PL=0
MOVL C01050 V=800.0 PL=0
MOVL C01051 V=800.0 PL=0
MOVL C01052 V=800.0 PL=0
MOVL C01053 V=800.0 PL=0
MOVL C01054 V=800.0 PL=0
MOVL C01055 V=800.0 PL=0
MOVL C01056 V=800.0 PL=0
MOVL C01057 V=800.0 PL=0
MOVL C01058 V=800.0 PL=0
MOVL C01059 V=800.0 PL=0
MOVL C01060 V=800.0 PL=0
MOVL C01061 V=800.0 PL=0
MOVL C01062 V=800.0 PL=0
MOVL C01063 V=800.0 PL=0
MOVL C01064 V=800.0 PL=0
MOVL C01065 V=800.0 PL=0
MOVL C01066 V=800.0 PL=0
MOVL C01067 V=800.0 PL=0
MOVL C01068 V=800.0 PL=0
MOVL C01069 V=800.0 PL=0
MOVL C01070 V=800.0 PL=0
MOVL C01071 V=800.0 PL=0
MOVL C01072 V=800.0 PL=0
MOVL C01073 V=800.0 PL=0
MOVL C01074 V=800.0 PL=0
MOVL C01075 V=800.0 PL=0
MOVL C01076 V=800.0 PL=0
MOVL C01077 V=800.0 PL=0
MOVL C01078 V=800.0 PL=0
MOVL C01079 V=800.0 PL=0
MOVL C01080 V=800.0 PL=0
MOVL C01081 V=800.0 PL=0
MOVL C01082 V=800.0 PL=0
MOVL C01083 V=800.0 PL=0
MOVL C01084 V=800.0 PL=0
MOVL C01085 V=800.0 PL=0
MOVL C01086 V=800.0 PL=0
MOVL C01087 V=800.0 PL=0
MOVL C01088 V=800.0 PL=0
MOVL C01089 V=800.0 PL=0
MOVL C01090 V=800.0 PL=0
MOVL C01091 V=800.0 PL=0
MOVL C01092 V=800.0 PL=0
MOVL C01093 V=800.0 PL=0
MOVL C01094 V=800.0 PL=0
MOVL C01095 V=800.0 PL=0
MOVL C01096 V=800.0 PL=0
MOVL C01097 V=800.0 PL=0
MOVL C01098 V=800.0 PL=0
MOVL C01099 V=800.0 PL=0
MOVL C01100 V=800.0 PL=0
MOVL C01101 V=800.0 PL=0
MOVL C01102 V=800.0 PL=0
MOVL C01103 V=800.0 PL=0
MOVL C01104 V=800.0 PL=0
MOVL C01105 V=800.0 PL=0
MOVL C01106 V=800.0 PL=0
MOVL C01107 V=800.0 PL=0
MOVL C01108 V=800.0 PL=0
MOVL C01109 V=800.0 PL=0
MOVL C01110 V=800.0 PL=0
MOVL C01111 V=800.0 PL=0
MOVL C01112 V=800.0 PL=0
MOVL C01113 V=800.0 PL=0
MOVL C01114 V=800.0 PL=0
MOVL C01115 V=800.0 PL=0
MOVL C01116 V=800.0 PL=0
MOVL C01117 V=800.0 PL=0
MOVL C01118 V=800.0 PL=0
MOVL C01119 V=800.0 PL=0
MOVL C01120 V=800.0 PL=0
MOVL C01121 V=800.0 PL=0
MOVL C01122 V=800.0 PL=0
MOVL C01123 V=800.0 PL=0
MOVL C01124 V=800.0 PL=0
MOVL C01125 V=800.0 PL=0
MOVL C01126 V=800.0 PL=0
MOVL C01127 V=800.0 PL=0
MOVL C01128 V=800.0 PL=0
MOVL C01129 V=800.0 PL=0
MOVL C01130 V=800.0 PL=0
MOVL C01131 V=800.0 PL=0
MOVL C01132 V=800.0 PL=0
MOVL C01133 V=800.0 PL=0
MOVL C01134 V=800.0 PL=0
MOVL C01135 V=800.0 PL=0
MOVL C01136 V=800.0 PL=0
MOVL C01137 V=800.0 PL=0
MOVL C01138 V=800.0 PL=0
MOVL C01139 V=800.0 PL=0
MOVL C01140 V=800.0 PL=0
MOVL C01141 V=800.0 PL=0
MOVL C01142 V=800.0 PL=0
MOVL C01143 V=800.0 PL=0
MOVL C01144 V=800.0 PL=0
MOVL C01145 V=800.0 PL=0
MOVL C01146 V=800.0 PL=0
MOVL C01147 V=800.0 PL=0
MOVL C01148 V=800.0 PL=0
MOVL C01149 V=800.0 PL=0
MOVL C01150 V=800.0 PL=0
MOVL C01151 V=800.0 PL=0
MOVL C01152 V=800.0 PL=0
MOVL C01153 V=800.0 PL=0
MOVL C01154 V=800.0 PL=0
MOVL C01155 V=800.0 PL=0
MOVL C01156 V=800.0 PL=0
MOVL C01157 V=800.0 PL=0
MOVL C01158 V=800.0 PL=0
MOVL C01159 V=800.0 PL=0
MOVL C01160 V=800.0 PL=0
MOVL C01161 V=800.0 PL=0
MOVL C01162 V=800.0 PL=0
MOVL C01163 V=800.0 PL=0
MOVL C01164 V=800.0 PL=0
MOVL C01165 V=800.0 PL=0
MOVL C01166 V=800.0 PL=0
MOVL C01167 V=800.0 PL=0
MOVL C01168 V=800.0 PL=0
MOVL C01169 V=800.0 PL=0
MOVL C01170 V=800.0 PL=0
MOVL C01171 V=800.0 PL=0
MOVL C01172 V=800.0 PL=0
MOVL C01173 V=800.0 PL=0
MOVL C01174 V=800.0 PL=0
MOVL C01175 V=800.0 PL=0
MOVL C01176 V=800.0 PL=0
MOVL C01177 V=800.0 PL=0
MOVL C01178 V=800.0 PL=0
MOVL C01179 V=800.0 PL=0
MOVL C01180 V=800.0 PL=0
MOVL C01181 V=800.0 PL=0
MOVL C01182 V=800.0 PL=0
MOVL C01183 V=800.0 PL=0
MOVL C01184 V=800.0 PL=0
MOVL C01185 V=800.0 PL=0
MOVL C01186 V=800.0 PL=0
MOVL C01187 V=800.0 PL=0
MOVL C01188 V=800.0 PL=0
MOVL C01189 V=800.0 PL=0
MOVL C01190 V=800.0 PL=0
MOVL C01191 V=800.0 PL=0
MOVL C01192 V=800.0 PL=0
MOVL C01193 V=800.0 PL=0
MOVL C01194 V=800.0 PL=0
MOVL C01195 V=800.0 PL=0
MOVL C01196 V=800.0 PL=0
MOVL C01197 V=800.0 PL=0
MOVL C01198 V=800.0 PL=0
MOVL C01199 V=800.0 PL=0
MOVL C01200 V=800.0 PL=0
MOVL C01201 V=800.0 PL=0
MOVL C01202 V=800.0 PL=0
MOVL C01203 V=800.0 PL=0
MOVL C01204 V=800.0 PL=0
MOVL C01205 V=800.0 PL=0
MOVL C01206 V=800.0 PL=0
MOVL C01207 V=800.0 PL=0
MOVL C01208 V=800.0 PL=0
MOVL C01209 V=800.0 PL=0
MOVL C01210 V=800.0 PL=0
MOVL C01211 V=800.0 PL=0
MOVL C01212 V=800.0 PL=0
MOVL C01213 V=800.0 PL=0
MOVL C01214 V=800.0 PL=0
MOVL C01215 V=800.0 PL=0
MOVL C01216 V=800.0 PL=0
MOVL C01217 V=800.0 PL=0
MOVL C01218 V=800.0 PL=0
MOVL C01219 V=800.0 PL=0
MOVL C01220 V=800.0 PL=0
MOVL C01221 V=800.0 PL=0
MOVL C01222 V=800.0 PL=0
MOVL C01223 V=800.0 PL=0
MOVL C01224 V=800.0 PL=0
MOVL C01225 V=800.0 PL=0
MOVL C01226 V=800.0 PL=0
MOVL C01227 V=800.0 PL=0
MOVL C01228 V=800.0 PL=0
MOVL C01229 V=800.0 PL=0
MOVL C01230 V=800.0 PL=0
MOVL C01231 V=800.0 PL=0
MOVL C01232 V=800.0 PL=0
MOVL C01233 V=800.0 PL=0
MOVL C01234 V=800.0 PL=0
MOVL C01235 V=800.0 PL=0
MOVL C01236 V=800.0 PL=0
MOVL C01237 V=800.0 PL=0
MOVL C01238 V=800.0 PL=0
MOVL C01239 V=800.0 PL=0
MOVL C01240 V=800.0 PL=0
MOVL C01241 V=800.0 PL=0
MOVL C01242 V=800.0 PL=0
MOVL C01243 V=800.0 PL=0
MOVL C01244 V=800.0 PL=0
MOVL C01245 V=800.0 PL=0
MOVL C01246 V=800.0 PL=0
MOVL C01247 V=800.0 PL=0
MOVL C01248 V=800.0 PL=0
MOVL C01249 V=800.0 PL=0
MOVL C01250 V=800.0 PL=0
MOVL C01251 V=800.0 PL=0
MOVL C01252 V=800.0 PL=0
MOVL C01253 V=800.0 PL=0
MOVL C01254 V=800.0 PL=0
MOVL C01255 V=800.0 PL=0
MOVL C01256 V=800.0 PL=0
MOVL C01257 V=800.0 PL=0
MOVL C01258 V=800.0 PL=0
MOVL C01259 V=800.0 PL=0
MOVL C01260 V=800.0 PL=0
MOVL C01261 V=800.0 PL=0
MOVL C01262 V=800.0 PL=0
MOVL C01263 V=800.0 PL=0
MOVL C01264 V=800.0 PL=0
MOVL C01265 V=800.0 PL=0
MOVL C01266 V=800.0 PL=0
MOVL C01267 V=800.0 PL=0
MOVL C01268 V=800.0 PL=0
MOVL C01269 V=800.0 PL=0
MOVL C01270 V=800.0 PL=0
MOVL C01271 V=800.0 PL=0
MOVL C01272 V=800.0 PL=0
MOVL C01273 V=800.0 PL=0
MOVL C01274 V=800.0 PL=0
MOVL C01275 V=800.0 PL=0
MOVL C01276 V=800.0 PL=0
MOVL C01277 V=800.0 PL=0
MOVL C01278 V=800.0 PL=0
MOVL C01279 V=800.0 PL=0
MOVL C01280 V=800.0 PL=0
MOVL C01281 V=800.0 PL=0
MOVL C01282 V=800.0 PL=0
MOVL C01283 V=800.0 PL=0
MOVL C01284 V=800.0 PL=0
MOVL C01285 V=800.0 PL=0
MOVL C01286 V=800.0 PL=0
MOVL C01287 V=800.0 PL=0
MOVL C01288 V=800.0 PL=0
MOVL C01289 V=800.0 PL=0
MOVL C01290 V=800.0 PL=0
MOVL C01291 V=800.0 PL=0
MOVL C01292 V=800.0 PL=0
MOVL C01293 V=800.0 PL=0
MOVL C01294 V=800.0 PL=0
MOVL C01295 V=800.0 PL=0
MOVL C01296 V=800.0 PL=0
MOVL C01297 V=800.0 PL=0
MOVL C01298 V=800.0 PL=0
MOVL C01299 V=800.0 PL=0
MOVL C01300 V=800.0 PL=0
MOVL C01301 V=800.0 PL=0
MOVL C01302 V=800.0 PL=0
MOVL C01303 V=800.0 PL=0
MOVL C01304 V=800.0 PL=0
MOVL C01305 V=800.0 PL=0
MOVL C01306 V=800.0 PL=0
MOVL C01307 V=800.0 PL=0
MOVL C01308 V=800.0 PL=0
MOVL C01309 V=800.0 PL=0
MOVL C01310 V=800.0 PL=0
MOVL C01311 V=800.0 PL=0
MOVL C01312 V=800.0 PL=0
MOVL C01313 V=800.0 PL=0
MOVL C01314 V=800.0 PL=0
MOVL C01315 V=800.0 PL=0
MOVL C01316 V=800.0 PL=0
MOVL C01317 V=800.0 PL=0
MOVL C01318 V=800.0 PL=0
MOVL C01319 V=800.0 PL=0
MOVL C01320 V=800.0 PL=0
MOVL C01321 V=800.0 PL=0
MOVL C01322 V=800.0 PL=0
MOVL C01323 V=800.0 PL=0
MOVL C01324 V=800.0 PL=0
MOVL C01325 V=800.0 PL=0
MOVL C01326 V=800.0 PL=0
MOVL C01327 V=800.0 PL=0
MOVL C01328 V=800.0 PL=0
MOVL C01329 V=800.0 PL=0
MOVL C01330 V=800.0 PL=0
MOVL C01331 V=800.0 PL=0
MOVL C01332 V=800.0 PL=0
MOVL C01333 V=800.0 PL=0
MOVL C01334 V=800.0 PL=0
MOVL C01335 V=800.0 PL=0
MOVL C01336 V=800.0 PL=0
MOVL C01337 V=800.0 PL=0
MOVL C01338 V=800.0 PL=0
MOVL C01339 V=800.0 PL=0
MOVL C01340 V=800.0 PL=0
MOVL C01341 V=800.0 PL=0
MOVL C01342 V=800.0 PL=0
MOVL C01343 V=800.0 PL=0
MOVL C01344 V=800.0 PL=0
MOVL C01345 V=800.0 PL=0
MOVL C01346 V=800.0 PL=0
MOVL C01347 V=800.0 PL=0
MOVL C01348 V=800.0 PL=0
MOVL C01349 V=800.0 PL=0
MOVL C01350 V=800.0 PL=0
MOVL C01351 V=800.0 PL=0
MOVL C01352 V=800.0 PL=0
MOVL C01353 V=800.0 PL=0
MOVL C01354 V=800.0 PL=0
MOVL C01355 V=800.0 PL=0
MOVL C01356 V=800.0 PL=0
MOVL C01357 V=800.0 PL=0
MOVL C01358 V=800.0 PL=0
MOVL C01359 V=800.0 PL=0
MOVL C01360 V=800.0 PL=0
MOVL C01361 V=800.0 PL=0
MOVL C01362 V=800.0 PL=0
MOVL C01363 V=800.0 PL=0
MOVL C01364 V=800.0 PL=0
MOVL C01365 V=800.0 PL=0
MOVL C01366 V=800.0 PL=0
MOVL C01367 V=800.0 PL=0
MOVL C01368 V=800.0 PL=0
MOVL C01369 V=800.0 PL=0
MOVL C01370 V=800.0 PL=0
MOVL C01371 V=800.0 PL=0
MOVL C01372 V=800.0 PL=0
MOVL C01373 V=800.0 PL=0
MOVL C01374 V=800.0 PL=0
MOVL C01375 V=800.0 PL=0
MOVL C01376 V=800.0 PL=0
MOVL C01377 V=800.0 PL=0
MOVL C01378 V=800.0 PL=0
MOVL C01379 V=800.0 PL=0
MOVL C01380 V=800.0 PL=0
MOVL C01381 V=800.0 PL=0
MOVL C01382 V=800.0 PL=0
MOVL C01383 V=800.0 PL=0
MOVL C01384 V=800.0 PL=0
MOVL C01385 V=800.0 PL=0
MOVL C01386 V=800.0 PL=0
MOVL C01387 V=800.0 PL=0
MOVL C01388 V=800.0 PL=0
MOVL C01389 V=800.0 PL=0
MOVL C01390 V=800.0 PL=0
MOVL C01391 V=800.0 PL=0
MOVL C01392 V=800.0 PL=0
MOVL C01393 V=800.0 PL=0
MOVL C01394 V=800.0 PL=0
MOVL C01395 V=800.0 PL=0
MOVL C01396 V=800.0 PL=0
MOVL C01397 V=800.0 PL=0
MOVL C01398 V=800.0 PL=0
MOVL C01399 V=800.0 PL=0
MOVL C01400 V=800.0 PL=0
MOVL C01401 V=800.0 PL=0
MOVL C01402 V=800.0 PL=0
MOVL C01403 V=800.0 PL=0
MOVL C01404 V=800.0 PL=0
MOVL C01405 V=800.0 PL=0
MOVL C01406 V=800.0 PL=0
MOVL C01407 V=800.0 PL=0
MOVL C01408 V=800.0 PL=0
MOVL C01409 V=800.0 PL=0
MOVL C01410 V=800.0 PL=0
MOVL C01411 V=800.0 PL=0
MOVL C01412 V=800.0 PL=0
MOVL C01413 V=800.0 PL=0
MOVL C01414 V=800.0 PL=0
MOVL C01415 V=800.0 PL=0
MOVL C01416 V=800.0 PL=0
MOVL C01417 V=800.0 PL=0
MOVL C01418 V=800.0 PL=0
MOVL C01419 V=800.0 PL=0
MOVL C01420 V=800.0 PL=0
MOVL C01421 V=800.0 PL=0
MOVL C01422 V=800.0 PL=0
MOVL C01423 V=800.0 PL=0
MOVL C01424 V=800.0 PL=0
MOVL C01425 V=800.0 PL=0
MOVL C01426 V=800.0 PL=0
MOVL C01427 V=800.0 PL=0
MOVL C01428 V=800.0 PL=0
MOVL C01429 V=800.0 PL=0
MOVL C01430 V=800.0 PL=0
MOVL C01431 V=800.0 PL=0
MOVL C01432 V=800.0 PL=0
MOVL C01433 V=800.0 PL=0
MOVL C01434 V=800.0 PL=0
MOVL C01435 V=800.0 PL=0
MOVL C01436 V=800.0 PL=0
MOVL C01437 V=800.0 PL=0
MOVL C01438 V=800.0 PL=0
MOVL C01439 V=800.0 PL=0
MOVL C01440 V=800.0 PL=0
MOVL C01441 V=800.0 PL=0
MOVL C01442 V=800.0 PL=0
MOVL C01443 V=800.0 PL=0
MOVL C01444 V=800.0 PL=0
MOVL C01445 V=800.0 PL=0
MOVL C01446 V=800.0 PL=0
MOVL C01447 V=800.0 PL=0
MOVL C01448 V=800.0 PL=0
MOVL C01449 V=800.0 PL=0
MOVL C01450 V=800.0 PL=0
MOVL C01451 V=800.0 PL=0
MOVL C01452 V=800.0 PL=0
MOVL C01453 V=800.0 PL=0
MOVL C01454 V=800.0 PL=0
MOVL C01455 V=800.0 PL=0
MOVL C01456 V=800.0 PL=0
MOVL C01457 V=800.0 PL=0
MOVL C01458 V=800.0 PL=0
MOVL C01459 V=800.0 PL=0
MOVL C01460 V=800.0 PL=0
MOVL C01461 V=800.0 PL=0
MOVL C01462 V=800.0 PL=0
MOVL C01463 V=800.0 PL=0
MOVL C01464 V=800.0 PL=0
MOVL C01465 V=800.0 PL=0
MOVL C01466 V=800.0 PL=0
MOVL C01467 V=800.0 PL=0
MOVL C01468 V=800.0 PL=0
MOVL C01469 V=800.0 PL=0
MOVL C01470 V=800.0 PL=0
MOVL C01471 V=800.0 PL=0
MOVL C01472 V=800.0 PL=0
MOVL C01473 V=800.0 PL=0
MOVL C01474 V=800.0 PL=0
MOVL C01475 V=800.0 PL=0
MOVL C01476 V=800.0 PL=0
MOVL C01477 V=800.0 PL=0
MOVL C01478 V=800.0 PL=0
MOVL C01479 V=800.0 PL=0
MOVL C01480 V=800.0 PL=0
MOVL C01481 V=800.0 PL=0
MOVL C01482 V=800.0 PL=0
MOVL C01483 V=800.0 PL=0
MOVL C01484 V=800.0 PL=0
MOVL C01485 V=800.0 PL=0
MOVL C01486 V=800.0 PL=0
MOVL C01487 V=800.0 PL=0
MOVL C01488 V=800.0 PL=0
MOVL C01489 V=800.0 PL=0
MOVL C01490 V=800.0 PL=0
MOVL C01491 V=800.0 PL=0
MOVL C01492 V=800.0 PL=0
MOVL C01493 V=800.0 PL=0
MOVL C01494 V=800.0 PL=0
MOVL C01495 V=800.0 PL=0
MOVL C01496 V=800.0 PL=0
MOVL C01497 V=800.0 PL=0
MOVL C01498 V=800.0 PL=0
MOVL C01499 V=800.0 PL=0
MOVL C01500 V=800.0 PL=0
MOVL C01501 V=800.0 PL=0
MOVL C01502 V=800.0 PL=0
MOVL C01503 V=800.0 PL=0
MOVL C01504 V=800.0 PL=0
MOVL C01505 V=800.0 PL=0
MOVL C01506 V=800.0 PL=0
MOVL C01507 V=800.0 PL=0
MOVL C01508 V=800.0 PL=0
MOVL C01509 V=800.0 PL=0
MOVL C01510 V=800.0 PL=0
MOVL C01511 V=800.0 PL=0
MOVL C01512 V=800.0 PL=0
MOVL C01513 V=800.0 PL=0
MOVL C01514 V=800.0 PL=0
MOVL C01515 V=800.0 PL=0
MOVL C01516 V=800.0 PL=0
MOVL C01517 V=800.0 PL=0
MOVL C01518 V=800.0 PL=0
MOVL C01519 V=800.0 PL=0
MOVL C01520 V=800.0 PL=0
MOVL C01521 V=800.0 PL=0
MOVL C01522 V=800.0 PL=0
MOVL C01523 V=800.0 PL=0
MOVL C01524 V=800.0 PL=0
MOVL C01525 V=800.0 PL=0
MOVL C01526 V=800.0 PL=0
MOVL C01527 V=800.0 PL=0
MOVL C01528 V=800.0 PL=0
MOVL C01529 V=800.0 PL=0
MOVL C01530 V=800.0 PL=0
MOVL C01531 V=800.0 PL=0
MOVL C01532 V=800.0 PL=0
MOVL C01533 V=800.0 PL=0
MOVL C01534 V=800.0 PL=0
MOVL C01535 V=800.0 PL=0
MOVL C01536 V=800.0 PL=0
MOVL C01537 V=800.0 PL=0
MOVL C01538 V=800.0 PL=0
MOVL C01539 V=800.0 PL=0
MOVL C01540 V=800.0 PL=0
MOVL C01541 V=800.0 PL=0
MOVL C01542 V=800.0 PL=0
MOVL C01543 V=800.0 PL=0
MOVL C01544 V=800.0 PL=0
MOVL C01545 V=800.0 PL=0
MOVL C01546 V=800.0 PL=0
MOVL C01547 V=800.0 PL=0
MOVL C01548 V=800.0 PL=0
MOVL C01549 V=800.0 PL=0
MOVL C01550 V=800.0 PL=0
MOVL C01551 V=800.0 PL=0
MOVL C01552 V=800.0 PL=0
MOVL C01553 V=800.0 PL=0
MOVL C01554 V=800.0 PL=0
MOVL C01555 V=800.0 PL=0
MOVL C01556 V=800.0 PL=0
MOVL C01557 V=800.0 PL=0
MOVL C01558 V=800.0 PL=0
MOVL C01559 V=800.0 PL=0
MOVL C01560 V=800.0 PL=0
MOVL C01561 V=800.0 PL=0
MOVL C01562 V=800.0 PL=0
MOVL C01563 V=800.0 PL=0
MOVL C01564 V=800.0 PL=0
MOVL C01565 V=800.0 PL=0
MOVL C01566 V=800.0 PL=0
MOVL C01567 V=800.0 PL=0
MOVL C01568 V=800.0 PL=0
MOVL C01569 V=800.0 PL=0
MOVL C01570 V=800.0 PL=0
MOVL C01571 V=800.0 PL=0
MOVL C01572 V=800.0 PL=0
MOVL C01573 V=800.0 PL=0
MOVL C01574 V=800.0 PL=0
MOVL C01575 V=800.0 PL=0
MOVL C01576 V=800.0 PL=0
MOVL C01577 V=800.0 PL=0
MOVL C01578 V=800.0 PL=0
MOVL C01579 V=800.0 PL=0
MOVL C01580 V=800.0 PL=0
MOVL C01581 V=800.0 PL=0
MOVL C01582 V=800.0 PL=0
MOVL C01583 V=800.0 PL=0
MOVL C01584 V=800.0 PL=0
MOVL C01585 V=800.0 PL=0
MOVL C01586 V=800.0 PL=0
MOVL C01587 V=800.0 PL=0
MOVL C01588 V=800.0 PL=0
MOVL C01589 V=800.0 PL=0
MOVL C01590 V=800.0 PL=0
MOVL C01591 V=800.0 PL=0
MOVL C01592 V=800.0 PL=0
MOVL C01593 V=800.0 PL=0
MOVL C01594 V=800.0 PL=0
MOVL C01595 V=800.0 PL=0
MOVL C01596 V=800.0 PL=0
MOVL C01597 V=800.0 PL=0
MOVL C01598 V=800.0 PL=0
MOVL C01599 V=800.0 PL=0
MOVL C01600 V=800.0 PL=0
MOVL C01601 V=800.0 PL=0
MOVL C01602 V=800.0 PL=0
MOVL C01603 V=800.0 PL=0
MOVL C01604 V=800.0 PL=0
MOVL C01605 V=800.0 PL=0
MOVL C01606 V=800.0 PL=0
MOVL C01607 V=800.0 PL=0
MOVL C01608 V=800.0 PL=0
MOVL C01609 V=800.0 PL=0
MOVL C01610 V=800.0 PL=0
MOVL C01611 V=800.0 PL=0
MOVL C01612 V=800.0 PL=0
MOVL C01613 V=800.0 PL=0
MOVL C01614 V=800.0 PL=0
MOVL C01615 V=800.0 PL=0
MOVL C01616 V=800.0 PL=0
MOVL C01617 V=800.0 PL=0
MOVL C01618 V=800.0 PL=0
MOVL C01619 V=800.0 PL=0
MOVL C01620 V=800.0 PL=0
MOVL C01621 V=800.0 PL=0
MOVL C01622 V=800.0 PL=0
MOVL C01623 V=800.0 PL=0
MOVL C01624 V=800.0 PL=0
MOVL C01625 V=800.0 PL=0
MOVL C01626 V=800.0 PL=0
MOVL C01627 V=800.0 PL=0
MOVL C01628 V=800.0 PL=0
MOVL C01629 V=800.0 PL=0
MOVL C01630 V=800.0 PL=0
MOVL C01631 V=800.0 PL=0
MOVL C01632 V=800.0 PL=0
MOVL C01633 V=800.0 PL=0
MOVL C01634 V=800.0 PL=0
MOVL C01635 V=800.0 PL=0
MOVL C01636 V=800.0 PL=0
MOVL C01637 V=800.0 PL=0
MOVL C01638 V=800.0 PL=0
MOVL C01639 V=800.0 PL=0
MOVL C01640 V=800.0 PL=0
MOVL C01641 V=800.0 PL=0
MOVL C01642 V=800.0 PL=0
MOVL C01643 V=800.0 PL=0
MOVL C01644 V=800.0 PL=0
MOVL C01645 V=800.0 PL=0
MOVL C01646 V=800.0 PL=0
MOVL C01647 V=800.0 PL=0
MOVL C01648 V=800.0 PL=0
MOVL C01649 V=800.0 PL=0
MOVL C01650 V=800.0 PL=0
MOVL C01651 V=800.0 PL=0
MOVL C01652 V=800.0 PL=0
MOVL C01653 V=800.0 PL=0
MOVL C01654 V=800.0 PL=0
MOVL C01655 V=800.0 PL=0
MOVL C01656 V=800.0 PL=0
MOVL C01657 V=800.0 PL=0
MOVL C01658 V=800.0 PL=0
MOVL C01659 V=800.0 PL=0
MOVL C01660 V=800.0 PL=0
MOVL C01661 V=800.0 PL=0
MOVL C01662 V=800.0 PL=0
MOVL C01663 V=800.0 PL=0
MOVL C01664 V=800.0 PL=0
MOVL C01665 V=800.0 PL=0
MOVL C01666 V=800.0 PL=0
MOVL C01667 V=800.0 PL=0
MOVL C01668 V=800.0 PL=0
MOVL C01669 V=800.0 PL=0
MOVL C01670 V=800.0 PL=0
MOVL C01671 V=800.0 PL=0
MOVL C01672 V=800.0 PL=0
MOVL C01673 V=800.0 PL=0
MOVL C01674 V=800.0 PL=0
MOVL C01675 V=800.0 PL=0
MOVL C01676 V=800.0 PL=0
MOVL C01677 V=800.0 PL=0
MOVL C01678 V=800.0 PL=0
MOVL C01679 V=800.0 PL=0
MOVL C01680 V=800.0 PL=0
MOVL C01681 V=800.0 PL=0
MOVL C01682 V=800.0 PL=0
MOVL C01683 V=800.0 PL=0
MOVL C01684 V=800.0 PL=0
MOVL C01685 V=800.0 PL=0
MOVL C01686 V=800.0 PL=0
MOVL C01687 V=800.0 PL=0
MOVL C01688 V=800.0 PL=0
MOVL C01689 V=800.0 PL=0
MOVL C01690 V=800.0 PL=0
MOVL C01691 V=800.0 PL=0
MOVL C01692 V=800.0 PL=0
MOVL C01693 V=800.0 PL=0
MOVL C01694 V=800.0 PL=0
MOVL C01695 V=800.0 PL=0
MOVL C01696 V=800.0 PL=0
MOVL C01697 V=800.0 PL=0
MOVL C01698 V=800.0 PL=0
MOVL C01699 V=800.0 PL=0
MOVL C01700 V=800.0 PL=0
MOVL C01701 V=800.0 PL=0
MOVL C01702 V=800.0 PL=0
MOVL C01703 V=800.0 PL=0
MOVL C01704 V=800.0 PL=0
MOVL C01705 V=800.0 PL=0
MOVL C01706 V=800.0 PL=0
MOVL C01707 V=800.0 PL=0
MOVL C01708 V=800.0 PL=0
MOVL C01709 V=800.0 PL=0
MOVL C01710 V=800.0 PL=0
MOVL C01711 V=800.0 PL=0
MOVL C01712 V=800.0 PL=0
MOVL C01713 V=800.0 PL=0
MOVL C01714 V=800.0 PL=0
MOVL C01715 V=800.0 PL=0
MOVL C01716 V=800.0 PL=0
MOVL C01717 V=800.0 PL=0
MOVL C01718 V=800.0 PL=0
MOVL C01719 V=800.0 PL=0
MOVL C01720 V=800.0 PL=0
MOVL C01721 V=800.0 PL=0
MOVL C01722 V=800.0 PL=0
MOVL C01723 V=800.0 PL=0
MOVL C01724 V=800.0 PL=0
MOVL C01725 V=800.0 PL=0
MOVL C01726 V=800.0 PL=0
MOVL C01727 V=800.0 PL=0
MOVL C01728 V=800.0 PL=0
MOVL C01729 V=800.0 PL=0
MOVL C01730 V=800.0 PL=0
MOVL C01731 V=800.0 PL=0
MOVL C01732 V=800.0 PL=0
MOVL C01733 V=800.0 PL=0
MOVL C01734 V=800.0 PL=0
MOVL C01735 V=800.0 PL=0
MOVL C01736 V=800.0 PL=0
MOVL C01737 V=800.0 PL=0
MOVL C01738 V=800.0 PL=0
MOVL C01739 V=800.0 PL=0
MOVL C01740 V=800.0 PL=0
MOVL C01741 V=800.0 PL=0
MOVL C01742 V=800.0 PL=0
MOVL C01743 V=800.0 PL=0
MOVL C01744 V=800.0 PL=0
MOVL C01745 V=800.0 PL=0
MOVL C01746 V=800.0 PL=0
MOVL C01747 V=800.0 PL=0
MOVL C01748 V=800.0 PL=0
MOVL C01749 V=800.0 PL=0
MOVL C01750 V=800.0 PL=0
MOVL C01751 V=800.0 PL=0
MOVL C01752 V=800.0 PL=0
MOVL C01753 V=800.0 PL=0
MOVL C01754 V=800.0 PL=0
MOVL C01755 V=800.0 PL=0
MOVL C01756 V=800.0 PL=0
MOVL C01757 V=800.0 PL=0
MOVL C01758 V=800.0 PL=0
MOVL C01759 V=800.0 PL=0
MOVL C01760 V=800.0 PL=0
MOVL C01761 V=800.0 PL=0
MOVL C01762 V=800.0 PL=0
MOVL C01763 V=800.0 PL=0
MOVL C01764 V=800.0 PL=0
MOVL C01765 V=800.0 PL=0
MOVL C01766 V=800.0 PL=0
MOVL C01767 V=800.0 PL=0
MOVL C01768 V=800.0 PL=0
MOVL C01769 V=800.0 PL=0
MOVL C01770 V=800.0 PL=0
MOVL C01771 V=800.0 PL=0
MOVL C01772 V=800.0 PL=0
MOVL C01773 V=800.0 PL=0
MOVL C01774 V=800.0 PL=0
MOVL C01775 V=800.0 PL=0
MOVL C01776 V=800.0 PL=0
MOVL C01777 V=800.0 PL=0
MOVL C01778 V=800.0 PL=0
MOVL C01779 V=800.0 PL=0
MOVL C01780 V=800.0 PL=0
MOVL C01781 V=800.0 PL=0
MOVL C01782 V=800.0 PL=0
MOVL C01783 V=800.0 PL=0
MOVL C01784 V=800.0 PL=0
MOVL C01785 V=800.0 PL=0
MOVL C01786 V=800.0 PL=0
MOVL C01787 V=800.0 PL=0
MOVL C01788 V=800.0 PL=0
MOVL C01789 V=800.0 PL=0
MOVL C01790 V=800.0 PL=0
MOVL C01791 V=800.0 PL=0
MOVL C01792 V=800.0 PL=0
MOVL C01793 V=800.0 PL=0
MOVL C01794 V=800.0 PL=0
MOVL C01795 V=800.0 PL=0
MOVL C01796 V=800.0 PL=0
MOVL C01797 V=800.0 PL=0
MOVL C01798 V=800.0 PL=0
MOVL C01799 V=800.0 PL=0
MOVL C01800 V=800.0 PL=0
MOVL C01801 V=800.0 PL=0
MOVL C01802 V=800.0 PL=0
MOVL C01803 V=800.0 PL=0
MOVL C01804 V=800.0 PL=0
MOVL C01805 V=800.0 PL=0
MOVL C01806 V=800.0 PL=0
MOVL C01807 V=800.0 PL=0
MOVL C01808 V=800.0 PL=0
MOVL C01809 V=800.0 PL=0
MOVL C01810 V=800.0 PL=0
MOVL C01811 V=800.0 PL=0
MOVL C01812 V=800.0 PL=0
MOVL C01813 V=800.0 PL=0
MOVL C01814 V=800.0 PL=0
MOVL C01815 V=800.0 PL=0
MOVL C01816 V=800.0 PL=0
MOVL C01817 V=800.0 PL=0
MOVL C01818 V=800.0 PL=0
MOVL C01819 V=800.0 PL=0
MOVL C01820 V=800.0 PL=0
MOVL C01821 V=800.0 PL=0
MOVL C01822 V=800.0 PL=0
MOVL C01823 V=800.0 PL=0
MOVL C01824 V=800.0 PL=0
MOVL C01825 V=800.0 PL=0
MOVL C01826 V=800.0 PL=0
MOVL C01827 V=800.0 PL=0
MOVL C01828 V=800.0 PL=0
MOVL C01829 V=800.0 PL=0
MOVL C01830 V=800.0 PL=0
MOVL C01831 V=800.0 PL=0
MOVL C01832 V=800.0 PL=0
MOVL C01833 V=800.0 PL=0
MOVL C01834 V=800.0 PL=0
MOVL C01835 V=800.0 PL=0
MOVL C01836 V=800.0 PL=0
MOVL C01837 V=800.0 PL=0
MOVL C01838 V=800.0 PL=0
MOVL C01839 V=800.0 PL=0
MOVL C01840 V=800.0 PL=0
MOVL C01841 V=800.0 PL=0
MOVL C01842 V=800.0 PL=0
MOVL C01843 V=800.0 PL=0
MOVL C01844 V=800.0 PL=0
MOVL C01845 V=800.0 PL=0
MOVL C01846 V=800.0 PL=0
MOVL C01847 V=800.0 PL=0
MOVL C01848 V=800.0 PL=0
MOVL C01849 V=800.0 PL=0
MOVL C01850 V=800.0 PL=0
MOVL C01851 V=800.0 PL=0
MOVL C01852 V=800.0 PL=0
MOVL C01853 V=800.0 PL=0
MOVL C01854 V=800.0 PL=0
MOVL C01855 V=800.0 PL=0
MOVL C01856 V=800.0 PL=0
MOVL C01857 V=800.0 PL=0
MOVL C01858 V=800.0 PL=0
MOVL C01859 V=800.0 PL=0
MOVL C01860 V=800.0 PL=0
MOVL C01861 V=800.0 PL=0
MOVL C01862 V=800.0 PL=0
MOVL C01863 V=800.0 PL=0
MOVL C01864 V=800.0 PL=0
MOVL C01865 V=800.0 PL=0
MOVL C01866 V=800.0 PL=0
MOVL C01867 V=800.0 PL=0
MOVL C01868 V=800.0 PL=0
MOVL C01869 V=800.0 PL=0
MOVL C01870 V=800.0 PL=0
MOVL C01871 V=800.0 PL=0
MOVL C01872 V=800.0 PL=0
MOVL C01873 V=800.0 PL=0
MOVL C01874 V=800.0 PL=0
MOVL C01875 V=800.0 PL=0
MOVL C01876 V=800.0 PL=0
MOVL C01877 V=800.0 PL=0
MOVL C01878 V=800.0 PL=0
MOVL C01879 V=800.0 PL=0
MOVL C01880 V=800.0 PL=0
MOVL C01881 V=800.0 PL=0
MOVL C01882 V=800.0 PL=0
MOVL C01883 V=800.0 PL=0
MOVL C01884 V=800.0 PL=0
MOVL C01885 V=800.0 PL=0
MOVL C01886 V=800.0 PL=0
MOVL C01887 V=800.0 PL=0
MOVL C01888 V=800.0 PL=0
MOVL C01889 V=800.0 PL=0
MOVL C01890 V=800.0 PL=0
MOVL C01891 V=800.0 PL=0
MOVL C01892 V=800.0 PL=0
MOVL C01893 V=800.0 PL=0
MOVL C01894 V=800.0 PL=0
MOVL C01895 V=800.0 PL=0
MOVL C01896 V=800.0 PL=0
MOVL C01897 V=800.0 PL=0
MOVL C01898 V=800.0 PL=0
MOVL C01899 V=800.0 PL=0
MOVL C01900 V=800.0 PL=0
MOVL C01901 V=800.0 PL=0
MOVL C01902 V=800.0 PL=0
MOVL C01903 V=800.0 PL=0
MOVL C01904 V=800.0 PL=0
MOVL C01905 V=800.0 PL=0
MOVL C01906 V=800.0 PL=0
MOVL C01907 V=800.0 PL=0
MOVL C01908 V=800.0 PL=0
MOVL C01909 V=800.0 PL=0
MOVL C01910 V=800.0 PL=0
MOVL C01911 V=800.0 PL=0
MOVL C01912 V=800.0 PL=0
MOVL C01913 V=800.0 PL=0
MOVL C01914 V=800.0 PL=0
MOVL C01915 V=800.0 PL=0
MOVL C01916 V=800.0 PL=0
MOVL C01917 V=800.0 PL=0
MOVL C01918 V=800.0 PL=0
MOVL C01919 V=800.0 PL=0
MOVL C01920 V=800.0 PL=0
MOVL C01921 V=800.0 PL=0
MOVL C01922 V=800.0 PL=0
MOVL C01923 V=800.0 PL=0
MOVL C01924 V=800.0 PL=0
MOVL C01925 V=800.0 PL=0
MOVL C01926 V=800.0 PL=0
MOVL C01927 V=800.0 PL=0
MOVL C01928 V=800.0 PL=0
MOVL C01929 V=800.0 PL=0
MOVL C01930 V=800.0 PL=0
MOVL C01931 V=800.0 PL=0
MOVL C01932 V=800.0 PL=0
MOVL C01933 V=800.0 PL=0
MOVL C01934 V=800.0 PL=0
MOVL C01935 V=800.0 PL=0
MOVL C01936 V=800.0 PL=0
MOVL C01937 V=800.0 PL=0
MOVL C01938 V=800.0 PL=0
MOVL C01939 V=800.0 PL=0
MOVL C01940 V=800.0 PL=0
MOVL C01941 V=800.0 PL=0
MOVL C01942 V=800.0 PL=0
MOVL C01943 V=800.0 PL=0
MOVL C01944 V=800.0 PL=0
MOVL C01945 V=800.0 PL=0
MOVL C01946 V=800.0 PL=0
MOVL C01947 V=800.0 PL=0
MOVL C01948 V=800.0 PL=0
MOVL C01949 V=800.0 PL=0
MOVL C01950 V=800.0 PL=0
MOVL C01951 V=800.0 PL=0
MOVL C01952 V=800.0 PL=0
MOVL C01953 V=800.0 PL=0
MOVL C01954 V=800.0 PL=0
MOVL C01955 V=800.0 PL=0
MOVL C01956 V=800.0 PL=0
MOVL C01957 V=800.0 PL=0
MOVL C01958 V=800.0 PL=0
MOVL C01959 V=800.0 PL=0
MOVL C01960 V=800.0 PL=0
MOVL C01961 V=800.0 PL=0
MOVL C01962 V=800.0 PL=0
MOVL C01963 V=800.0 PL=0
MOVL C01964 V=800.0 PL=0
MOVL C01965 V=800.0 PL=0
MOVL C01966 V=800.0 PL=0
MOVL C01967 V=800.0 PL=0
MOVL C01968 V=800.0 PL=0
MOVL C01969 V=800.0 PL=0
MOVL C01970 V=800.0 PL=0
MOVL C01971 V=800.0 PL=0
MOVL C01972 V=800.0 PL=0
MOVL C01973 V=800.0 PL=0
MOVL C01974 V=800.0 PL=0
MOVL C01975 V=800.0 PL=0
MOVL C01976 V=800.0 PL=0
MOVL C01977 V=800.0 PL=0
MOVL C01978 V=800.0 PL=0
MOVL C01979 V=800.0 PL=0
MOVL C01980 V=800.0 PL=0
MOVL C01981 V=800.0 PL=0
MOVL C01982 V=800.0 PL=0
MOVL C01983 V=800.0 PL=0
MOVL C01984 V=800.0 PL=0
MOVL C01985 V=800.0 PL=0
MOVL C01986 V=800.0 PL=0
MOVL C01987 V=800.0 PL=0
MOVL C01988 V=800.0 PL=0
MOVL C01989 V=800.0 PL=0
MOVL C01990 V=800.0 PL=0
MOVL C01991 V=800.0 PL=0
MOVL C01992 V=800.0 PL=0
MOVL C01993 V=800.0 PL=0
MOVL C01994 V=800.0 PL=0
MOVL C01995 V=800.0 PL=0
MOVL C01996 V=800.0 PL=0
MOVL C01997 V=800.0 PL=0
MOVL C01998 V=800.0 PL=0
MOVL C01999 V=800.0 PL=0
MOVL C02000 V=800.0 PL=0
MOVL C02001 V=800.0 PL=0
MOVL C02002 V=800.0 PL=0
MOVL C02003 V=800.0 PL=0
MOVL C02004 V=800.0 PL=0
MOVL C02005 V=800.0 PL=0
MOVL C02006 V=800.0 PL=0
MOVL C02007 V=800.0 PL=0
MOVL C02008 V=800.0 PL=0
MOVL C02009 V=800.0 PL=0
MOVL C02010 V=800.0 PL=0
MOVL C02011 V=800.0 PL=0
MOVL C02012 V=800.0 PL=0
MOVL C02013 V=800.0 PL=0
MOVL C02014 V=800.0 PL=0
MOVL C02015 V=800.0 PL=0
MOVL C02016 V=800.0 PL=0
MOVL C02017 V=800.0 PL=0
MOVL C02018 V=800.0 PL=0
MOVL C02019 V=800.0 PL=0
MOVL C02020 V=800.0 PL=0
MOVL C02021 V=800.0 PL=0
MOVL C02022 V=800.0 PL=0
MOVL C02023 V=800.0 PL=0
MOVL C02024 V=800.0 PL=0
MOVL C02025 V=800.0 PL=0
MOVL C02026 V=800.0 PL=0
MOVL C02027 V=800.0 PL=0
MOVL C02028 V=800.0 PL=0
MOVL C02029 V=800.0 PL=0
MOVL C02030 V=800.0 PL=0
MOVL C02031 V=800.0 PL=0
MOVL C02032 V=800.0 PL=0
MOVL C02033 V=800.0 PL=0
MOVL C02034 V=800.0 PL=0
MOVL C02035 V=800.0 PL=0
MOVL C02036 V=800.0 PL=0
MOVL C02037 V=800.0 PL=0
